LIN {X 0,Y 418.256,Z 157.888,A -85,B 0,C 180,E1 -10109.163,E2 -10109.163} C_VEL
LIN {X 0,Y 418.233,Z 157.886,A -85,B 0,C 180,E1 -10112.53,E2 -10112.53} C_VEL
LIN {X 0,Y 418.25,Z 157.887,A -85,B 0,C 180,E1 -10114.842,E2 -10114.842} C_VEL
LIN {X 0,Y 418.23,Z 157.886,A -85,B 0,C 180,E1 -10118.445,E2 -10118.445} C_VEL
LIN {X 0,Y 418.219,Z 157.887,A -85,B 0,C 180,E1 -10122.236,E2 -10122.236} C_VEL
LIN {X 0,Y 418.238,Z 157.887,A -85,B 0,C 180,E1 -10125.108,E2 -10125.108} C_VEL
LIN {X 0,Y 418.219,Z 157.886,A -85,B 0,C 180,E1 -10127.764,E2 -10127.764} C_VEL
LIN {X 0,Y 418.198,Z 157.895,A -85,B 0,C 180,E1 -10130.629,E2 -10130.629} C_VEL
LIN {X 0,Y 418.221,Z 157.886,A -85,B 0,C 180,E1 -10133.973,E2 -10133.973} C_VEL
LIN {X 0,Y 418.231,Z 157.884,A -85,B 0,C 180,E1 -10137.47,E2 -10137.47} C_VEL
LIN {X 0,Y 418.261,Z 157.886,A -85,B 0,C 180,E1 -10140.898,E2 -10140.898} C_VEL
LIN {X 0,Y 418.242,Z 157.942,A -85,B 0,C 180,E1 -10143.423,E2 -10143.423} C_VEL
LIN {X 0,Y 418.819,Z 160.686,A -85,B 0,C 180,E1 -10144.132,E2 -10144.132} C_VEL
LIN {X 0,Y 420.946,Z 171.955,A -85,B 0,C 180,E1 -10146.675,E2 -10146.675} C_VEL
LIN {X 0,Y 420.228,Z 183.952,A -85,B 0,C 180,E1 -10149.182,E2 -10149.182} C_VEL
LIN {X 0,Y 419.697,Z 193.077,A -85,B 0,C 180,E1 -10151.036,E2 -10151.036} C_VEL
LIN {X 0,Y 420.352,Z 197.644,A -85,B 0,C 180,E1 -10151.195,E2 -10151.195} C_VEL
LIN {X 0,Y 423.589,Z 218.355,A -85,B 0,C 180,E1 -10151.71,E2 -10151.71} C_VEL
LIN {X 0,Y 422.515,Z 301.675,A -85,B 0,C 180,E1 -10153.2,E2 -10153.2} C_VEL
LIN {X 0,Y 422,Z 315.355,A -85,B 0,C 180,E1 -10153.646,E2 -10153.646} C_VEL
LIN {X 0,Y 421.401,Z 328.225,A -85,B 0,C 180,E1 -10154.275,E2 -10154.275} C_VEL
LIN {X 0,Y 420.651,Z 340.778,A -85,B 0,C 180,E1 -10155.114,E2 -10155.114} C_VEL
LIN {X 0,Y 419.944,Z 352.093,A -85,B 0,C 180,E1 -10156.089,E2 -10156.089} C_VEL
LIN {X 0,Y 419.366,Z 362.073,A -85,B 0,C 180,E1 -10157.17,E2 -10157.17} C_VEL
LIN {X 0,Y 418.661,Z 371.189,A -85,B 0,C 180,E1 -10158.378,E2 -10158.378} C_VEL
LIN {X 0,Y 418.066,Z 380.082,A -85,B 0,C 180,E1 -10159.832,E2 -10159.832} C_VEL
LIN {X 0,Y 417.587,Z 387.196,A -85,B 0,C 180,E1 -10161.287,E2 -10161.287} C_VEL
LIN {X 0,Y 417.292,Z 392.868,A -85,B 0,C 180,E1 -10162.742,E2 -10162.742} C_VEL
LIN {X 0,Y 417.127,Z 397.326,A -85,B 0,C 180,E1 -10164.197,E2 -10164.197} C_VEL
LIN {X 0,Y 417.115,Z 399.677,A -85,B 0,C 180,E1 -10165.166,E2 -10165.166} C_VEL
LIN {X 0,Y 417,Z 401.592,A -85,B 0,C 180,E1 -10166.134,E2 -10166.134} C_VEL
LIN {X 0,Y 416.985,Z 403.061,A -85,B 0,C 180,E1 -10167.101,E2 -10167.101} C_VEL
LIN {X 0,Y 417.031,Z 404.093,A -85,B 0,C 180,E1 -10168.068,E2 -10168.068} C_VEL
LIN {X 0,Y 416.983,Z 404.982,A -85,B 0,C 180,E1 -10169.999,E2 -10169.999} C_VEL
LIN {X 0,Y 416.993,Z 404.811,A -85,B 0,C 180,E1 -10170.965,E2 -10170.965} C_VEL
LIN {X 0,Y 417.03,Z 404.222,A -85,B 0,C 180,E1 -10171.93,E2 -10171.93} C_VEL
LIN {X 0,Y 417,Z 401.865,A -85,B 0,C 180,E1 -10173.864,E2 -10173.864} C_VEL
LIN {X 0,Y 417.158,Z 398.955,A -85,B 0,C 180,E1 -10175.316,E2 -10175.316} C_VEL
LIN {X 0,Y 417.245,Z 395.007,A -85,B 0,C 180,E1 -10176.77,E2 -10176.77} C_VEL
LIN {X 0,Y 417.536,Z 389.923,A -85,B 0,C 180,E1 -10178.225,E2 -10178.225} C_VEL
LIN {X 0,Y 417.921,Z 383.532,A -85,B 0,C 180,E1 -10179.68,E2 -10179.68} C_VEL
LIN {X 0,Y 418.465,Z 375.535,A -85,B 0,C 180,E1 -10181.135,E2 -10181.135} C_VEL
LIN {X 0,Y 419.313,Z 365.602,A -85,B 0,C 180,E1 -10182.584,E2 -10182.584} C_VEL
LIN {X 0,Y 419.963,Z 355.585,A -85,B 0,C 180,E1 -10183.754,E2 -10183.754} C_VEL
LIN {X 0,Y 420.694,Z 344.905,A -85,B 0,C 180,E1 -10184.758,E2 -10184.758} C_VEL
LIN {X 0,Y 421.389,Z 333.667,A -85,B 0,C 180,E1 -10185.6,E2 -10185.6} C_VEL
LIN {X 0,Y 422.192,Z 321.034,A -85,B 0,C 180,E1 -10186.313,E2 -10186.313} C_VEL
LIN {X 0,Y 422.754,Z 307.58,A -85,B 0,C 180,E1 -10186.85,E2 -10186.85} C_VEL
LIN {X 0,Y 423.111,Z 294.306,A -85,B 0,C 180,E1 -10187.177,E2 -10187.177} C_VEL
LIN {X 0,Y 423.985,Z 216.483,A -85,B 0,C 180,E1 -10188.568,E2 -10188.568} C_VEL
LIN {X 0,Y 420.139,Z 194.167,A -85,B 0,C 180,E1 -10189.181,E2 -10189.181} C_VEL
LIN {X 0,Y 419.921,Z 192.559,A -85,B 0,C 180,E1 -10189.275,E2 -10189.275} C_VEL
LIN {X 0,Y 421.094,Z 174.5,A -85,B 0,C 180,E1 -10192.964,E2 -10192.964} C_VEL
LIN {X 0,Y 420.573,Z 169.022,A -85,B 0,C 180,E1 -10194.166,E2 -10194.166} C_VEL
LIN {X 0,Y 418.252,Z 157.975,A -85,B 0,C 180,E1 -10196.777,E2 -10196.777} C_VEL
LIN {X 0,Y 418.23,Z 157.89,A -85,B 0,C 180,E1 -10200.272,E2 -10200.272} C_VEL
LIN {X 0,Y 418.226,Z 157.888,A -85,B 0,C 180,E1 -10203.677,E2 -10203.677} C_VEL
LIN {X 0,Y 418.226,Z 157.891,A -85,B 0,C 180,E1 -10207.224,E2 -10207.224} C_VEL
LIN {X 0,Y 418.2,Z 157.892,A -85,B 0,C 180,E1 -10210.866,E2 -10210.866} C_VEL
LIN {X 0,Y 418.194,Z 157.892,A -85,B 0,C 180,E1 -10213.726,E2 -10213.726} C_VEL
LIN {X 0,Y 418.19,Z 157.891,A -85,B 0,C 180,E1 -10216.446,E2 -10216.446} C_VEL
LIN {X 0,Y 418.198,Z 157.892,A -85,B 0,C 180,E1 -10219.132,E2 -10219.132} C_VEL
LIN {X 0,Y 418.225,Z 157.885,A -85,B 0,C 180,E1 -10222.774,E2 -10222.774} C_VEL
LIN {X 0,Y 418.222,Z 157.884,A -85,B 0,C 180,E1 -10226.32,E2 -10226.32} C_VEL
LIN {X 0,Y 418.227,Z 157.886,A -85,B 0,C 180,E1 -10229.726,E2 -10229.726} C_VEL
LIN {X 0,Y 418.198,Z 157.889,A -85,B 0,C 180,E1 -10233.015,E2 -10233.015} C_VEL
LIN {X 0,Y 418.244,Z 157.882,A -85,B 0,C 180,E1 -10236.216,E2 -10236.216} C_VEL
LIN {X 0,Y 418.237,Z 157.885,A -85,B 0,C 180,E1 -10239.336,E2 -10239.336} C_VEL
LIN {X 0,Y 418.267,Z 157.881,A -85,B 0,C 180,E1 -10242.395,E2 -10242.395} C_VEL
LIN {X 0,Y 418.284,Z 157.878,A -85,B 0,C 180,E1 -10245.402,E2 -10245.402} C_VEL
LIN {X 0,Y 418.299,Z 157.878,A -85,B 0,C 180,E1 -10248.368,E2 -10248.368} C_VEL
LIN {X 0,Y 418.453,Z 157.86,A -85,B 0,C 180,E1 -10252.278,E2 -10252.278} C_VEL
LIN {X 0,Y 418.485,Z 157.854,A -85,B 0,C 180,E1 -10254.216,E2 -10254.216} C_VEL
LIN {X 0,Y 418.523,Z 157.85,A -85,B 0,C 180,E1 -10258.075,E2 -10258.075} C_VEL
LIN {X 0,Y 418.466,Z 157.859,A -85,B 0,C 180,E1 -10260.962,E2 -10260.962} C_VEL
LIN {X 0,Y 418.46,Z 157.856,A -85,B 0,C 180,E1 -10262.888,E2 -10262.888} C_VEL
LIN {X 0,Y 418.45,Z 157.861,A -85,B 0,C 180,E1 -10266.682,E2 -10266.682} C_VEL
LIN {X 0,Y 418.311,Z 157.875,A -85,B 0,C 180,E1 -10269.672,E2 -10269.672} C_VEL
LIN {X 0,Y 418.332,Z 157.874,A -85,B 0,C 180,E1 -10273,E2 -10273} C_VEL
LIN {X 0,Y 418.298,Z 157.881,A -85,B 0,C 180,E1 -10276.735,E2 -10276.735} C_VEL
LIN {X 0,Y 418.256,Z 157.885,A -85,B 0,C 180,E1 -10279.79,E2 -10279.79} C_VEL
LIN {X 0,Y 418.214,Z 157.891,A -85,B 0,C 180,E1 -10282.737,E2 -10282.737} C_VEL
LIN {X 0,Y 418.204,Z 157.893,A -85,B 0,C 180,E1 -10285.908,E2 -10285.908} C_VEL
LIN {X 0,Y 418.269,Z 158.07,A -85,B 0,C 180,E1 -10289.645,E2 -10289.645} C_VEL
LIN {X 0,Y 420.353,Z 168.154,A -85,B 0,C 180,E1 -10292.061,E2 -10292.061} C_VEL
LIN {X 0,Y 420.567,Z 172.653,A -85,B 0,C 180,E1 -10293.062,E2 -10293.062} C_VEL
LIN {X 0,Y 420.213,Z 181.073,A -85,B 0,C 180,E1 -10294.813,E2 -10294.813} C_VEL
LIN {X 0,Y 423.231,Z 196.278,A -85,B 0,C 180,E1 -10295.287,E2 -10295.287} C_VEL
LIN {X 0,Y 424.291,Z 202.854,A -85,B 0,C 180,E1 -10295.463,E2 -10295.463} C_VEL
LIN {X 0,Y 422.997,Z 288.987,A -85,B 0,C 180,E1 -10297.017,E2 -10297.017} C_VEL
LIN {X 0,Y 422.616,Z 302.178,A -85,B 0,C 180,E1 -10297.45,E2 -10297.45} C_VEL
LIN {X 0,Y 422.093,Z 314.233,A -85,B 0,C 180,E1 -10298.029,E2 -10298.029} C_VEL
LIN {X 0,Y 421.458,Z 325.771,A -85,B 0,C 180,E1 -10298.77,E2 -10298.77} C_VEL
LIN {X 0,Y 420.642,Z 337.831,A -85,B 0,C 180,E1 -10299.778,E2 -10299.778} C_VEL
LIN {X 0,Y 419.841,Z 348.696,A -85,B 0,C 180,E1 -10300.925,E2 -10300.925} C_VEL
LIN {X 0,Y 419.105,Z 358.292,A -85,B 0,C 180,E1 -10302.198,E2 -10302.198} C_VEL
LIN {X 0,Y 418.472,Z 366.391,A -85,B 0,C 180,E1 -10303.517,E2 -10303.517} C_VEL
LIN {X 0,Y 417.906,Z 374.069,A -85,B 0,C 180,E1 -10305.066,E2 -10305.066} C_VEL
LIN {X 0,Y 417.524,Z 380.328,A -85,B 0,C 180,E1 -10306.694,E2 -10306.694} C_VEL
LIN {X 0,Y 417.245,Z 385.249,A -85,B 0,C 180,E1 -10308.373,E2 -10308.373} C_VEL
LIN {X 0,Y 417.139,Z 387.376,A -85,B 0,C 180,E1 -10309.302,E2 -10309.302} C_VEL
LIN {X 0,Y 416.926,Z 389.978,A -85,B 0,C 180,E1 -10310.841,E2 -10310.841} C_VEL
LIN {X 0,Y 416.831,Z 391.652,A -85,B 0,C 180,E1 -10312.631,E2 -10312.631} C_VEL
LIN {X 0,Y 416.778,Z 392.031,A -85,B 0,C 180,E1 -10314.037,E2 -10314.037} C_VEL
LIN {X 0,Y 416.834,Z 391.349,A -85,B 0,C 180,E1 -10315.706,E2 -10315.706} C_VEL
LIN {X 0,Y 416.908,Z 389.362,A -85,B 0,C 180,E1 -10317.444,E2 -10317.444} C_VEL
LIN {X 0,Y 417.17,Z 385.931,A -85,B 0,C 180,E1 -10319.225,E2 -10319.225} C_VEL
LIN {X 0,Y 417.366,Z 381.677,A -85,B 0,C 180,E1 -10320.771,E2 -10320.771} C_VEL
LIN {X 0,Y 417.733,Z 375.554,A -85,B 0,C 180,E1 -10322.442,E2 -10322.442} C_VEL
LIN {X 0,Y 418.212,Z 367.784,A -85,B 0,C 180,E1 -10324.094,E2 -10324.094} C_VEL
LIN {X 0,Y 418.738,Z 359.673,A -85,B 0,C 180,E1 -10325.457,E2 -10325.457} C_VEL
LIN {X 0,Y 419.405,Z 350.387,A -85,B 0,C 180,E1 -10326.724,E2 -10326.724} C_VEL
LIN {X 0,Y 420.143,Z 339.8,A -85,B 0,C 180,E1 -10327.892,E2 -10327.892} C_VEL
LIN {X 0,Y 420.86,Z 328.814,A -85,B 0,C 180,E1 -10328.854,E2 -10328.854} C_VEL
LIN {X 0,Y 421.51,Z 316.491,A -85,B 0,C 180,E1 -10329.697,E2 -10329.697} C_VEL
LIN {X 0,Y 421.984,Z 304.982,A -85,B 0,C 180,E1 -10330.292,E2 -10330.292} C_VEL
LIN {X 0,Y 422.414,Z 292.048,A -85,B 0,C 180,E1 -10330.758,E2 -10330.758} C_VEL
LIN {X 0,Y 422.684,Z 275.71,A -85,B 0,C 180,E1 -10331.1,E2 -10331.1} C_VEL
LIN {X 0,Y 423.205,Z 232.959,A -85,B 0,C 180,E1 -10331.848,E2 -10331.848} C_VEL
LIN {X 0,Y 422.703,Z 227.158,A -85,B 0,C 180,E1 -10331.974,E2 -10331.974} C_VEL
LIN {X 0,Y 417.261,Z 206.531,A -85,B 0,C 180,E1 -10332.579,E2 -10332.579} C_VEL
LIN {X 0,Y 416.803,Z 202.658,A -85,B 0,C 180,E1 -10332.67,E2 -10332.67} C_VEL
LIN {X 0,Y 412.969,Z 181.704,A -85,B 0,C 180,E1 -10333.248,E2 -10333.248} C_VEL
LIN {X 0,Y 412.905,Z 180.585,A -85,B 0,C 180,E1 -10333.373,E2 -10333.373} C_VEL
LIN {X 0,Y 413.489,Z 170.534,A -85,B 0,C 180,E1 -10335.652,E2 -10335.652} C_VEL
LIN {X 0,Y 411.309,Z 158.9,A -85,B 0,C 180,E1 -10338.544,E2 -10338.544} C_VEL
LIN {X 0,Y 411.441,Z 158.734,A -85,B 0,C 180,E1 -10342.185,E2 -10342.185} C_VEL
LIN {X 0,Y 411.472,Z 158.731,A -85,B 0,C 180,E1 -10344.119,E2 -10344.119} C_VEL
LIN {X 0,Y 411.508,Z 158.726,A -85,B 0,C 180,E1 -10348.044,E2 -10348.044} C_VEL
LIN {X 0,Y 411.637,Z 158.71,A -85,B 0,C 180,E1 -10350.001,E2 -10350.001} C_VEL
LIN {X 0,Y 411.455,Z 158.729,A -85,B 0,C 180,E1 -10352.938,E2 -10352.938} C_VEL
LIN {X 0,Y 411.464,Z 158.731,A -85,B 0,C 180,E1 -10355.883,E2 -10355.883} C_VEL
LIN {X 0,Y 411.317,Z 158.746,A -85,B 0,C 180,E1 -10358.847,E2 -10358.847} C_VEL
LIN {X 0,Y 411.283,Z 158.753,A -85,B 0,C 180,E1 -10361.834,E2 -10361.834} C_VEL
LIN {X 0,Y 411.259,Z 158.754,A -85,B 0,C 180,E1 -10364.854,E2 -10364.854} C_VEL
LIN {X 0,Y 411.244,Z 158.756,A -85,B 0,C 180,E1 -10367.916,E2 -10367.916} C_VEL
LIN {X 0,Y 411.195,Z 158.765,A -85,B 0,C 180,E1 -10371.035,E2 -10371.035} C_VEL
LIN {X 0,Y 411.224,Z 158.757,A -85,B 0,C 180,E1 -10374.216,E2 -10374.216} C_VEL
LIN {X 0,Y 411.258,Z 158.756,A -85,B 0,C 180,E1 -10377.478,E2 -10377.478} C_VEL
LIN {X 0,Y 411.188,Z 158.766,A -85,B 0,C 180,E1 -10380.848,E2 -10380.848} C_VEL
LIN {X 0,Y 411.204,Z 158.761,A -85,B 0,C 180,E1 -10384.334,E2 -10384.334} C_VEL
LIN {X 0,Y 411.191,Z 158.761,A -85,B 0,C 180,E1 -10387.975,E2 -10387.975} C_VEL
LIN {X 0,Y 411.163,Z 158.768,A -85,B 0,C 180,E1 -10391.229,E2 -10391.229} C_VEL
LIN {X 0,Y 411.175,Z 158.767,A -85,B 0,C 180,E1 -10394.491,E2 -10394.491} C_VEL
LIN {X 0,Y 411.171,Z 158.766,A -85,B 0,C 180,E1 -10398.195,E2 -10398.195} C_VEL
LIN {X 0,Y 411.197,Z 158.766,A -85,B 0,C 180,E1 -10400.774,E2 -10400.774} C_VEL
LIN {X 0,Y 411.197,Z 158.767,A -85,B 0,C 180,E1 -10404.472,E2 -10404.472} C_VEL
LIN {X 0,Y 411.207,Z 158.762,A -85,B 0,C 180,E1 -10406.874,E2 -10406.874} C_VEL
LIN {X 0,Y 411.212,Z 158.763,A -85,B 0,C 180,E1 -10410.65,E2 -10410.65} C_VEL
LIN {X 0,Y 411.195,Z 158.761,A -85,B 0,C 180,E1 -10413.617,E2 -10413.617} C_VEL
LIN {X 0,Y 411.202,Z 158.761,A -85,B 0,C 180,E1 -10416.853,E2 -10416.853} C_VEL
LIN {X 0,Y 411.215,Z 158.763,A -85,B 0,C 180,E1 -10420.051,E2 -10420.051} C_VEL
LIN {X 0,Y 411.264,Z 158.752,A -85,B 0,C 180,E1 -10423.132,E2 -10423.132} C_VEL
LIN {X 0,Y 411.306,Z 158.747,A -85,B 0,C 180,E1 -10426.897,E2 -10426.897} C_VEL
LIN {X 0,Y 411.288,Z 158.754,A -85,B 0,C 180,E1 -10430.162,E2 -10430.162} C_VEL
LIN {X 0,Y 411.39,Z 158.737,A -85,B 0,C 180,E1 -10433.132,E2 -10433.132} C_VEL
LIN {X 0,Y 411.289,Z 158.749,A -85,B 0,C 180,E1 -10435.099,E2 -10435.099} C_VEL
LIN {X 0,Y 411.502,Z 158.727,A -85,B 0,C 180,E1 -10438.043,E2 -10438.043} C_VEL
LIN {X 0,Y 411.377,Z 158.738,A -85,B 0,C 180,E1 -10440.979,E2 -10440.979} C_VEL
LIN {X 0,Y 411.439,Z 158.731,A -85,B 0,C 180,E1 -10442.938,E2 -10442.938} C_VEL
LIN {X 0,Y 411.386,Z 158.737,A -85,B 0,C 180,E1 -10446.869,E2 -10446.869} C_VEL
LIN {X 0,Y 411.282,Z 158.754,A -85,B 0,C 180,E1 -10449.839,E2 -10449.839} C_VEL
LIN {X 0,Y 411.307,Z 158.749,A -85,B 0,C 180,E1 -10453.104,E2 -10453.104} C_VEL
LIN {X 0,Y 411.259,Z 158.754,A -85,B 0,C 180,E1 -10456.889,E2 -10456.889} C_VEL
LIN {X 0,Y 411.212,Z 158.76,A -85,B 0,C 180,E1 -10459.988,E2 -10459.988} C_VEL
LIN {X 0,Y 411.189,Z 158.767,A -85,B 0,C 180,E1 -10463.149,E2 -10463.149} C_VEL
LIN {X 0,Y 411.165,Z 158.765,A -85,B 0,C 180,E1 -10466.386,E2 -10466.386} C_VEL
LIN {X 0,Y 411.194,Z 158.762,A -85,B 0,C 180,E1 -10469.714,E2 -10469.714} C_VEL
LIN {X 0,Y 411.205,Z 158.766,A -85,B 0,C 180,E1 -10473.156,E2 -10473.156} C_VEL
LIN {X 0,Y 411.19,Z 158.764,A -85,B 0,C 180,E1 -10476.552,E2 -10476.552} C_VEL
LIN {X 0,Y 411.166,Z 158.765,A -85,B 0,C 180,E1 -10479.719,E2 -10479.719} C_VEL
LIN {X 0,Y 411.163,Z 158.768,A -85,B 0,C 180,E1 -10483.135,E2 -10483.135} C_VEL
LIN {X 0,Y 411.166,Z 158.764,A -85,B 0,C 180,E1 -10485.882,E2 -10485.882} C_VEL
LIN {X 0,Y 411.158,Z 158.766,A -85,B 0,C 180,E1 -10489.492,E2 -10489.492} C_VEL
LIN {X 0,Y 411.173,Z 158.765,A -85,B 0,C 180,E1 -10492.023,E2 -10492.023} C_VEL
LIN {X 0,Y 411.185,Z 158.764,A -85,B 0,C 180,E1 -10495.127,E2 -10495.127} C_VEL
LIN {X 0,Y 411.176,Z 158.769,A -85,B 0,C 180,E1 -10498.719,E2 -10498.719} C_VEL
LIN {X 0,Y 411.171,Z 158.769,A -85,B 0,C 180,E1 -10501.406,E2 -10501.406} C_VEL
LIN {X 0,Y 411.222,Z 158.886,A -85,B 0,C 180,E1 -10503.221,E2 -10503.221} C_VEL
LIN {X 0,Y 413.471,Z 170.32,A -85,B 0,C 180,E1 -10505.924,E2 -10505.924} C_VEL
LIN {X 0,Y 413.991,Z 173.4,A -85,B 0,C 180,E1 -10506.622,E2 -10506.622} C_VEL
LIN {X 0,Y 413.246,Z 184.945,A -85,B 0,C 180,E1 -10509.074,E2 -10509.074} C_VEL
LIN {X 0,Y 412.771,Z 193.03,A -85,B 0,C 180,E1 -10510.738,E2 -10510.738} C_VEL
LIN {X 0,Y 413.463,Z 197.805,A -85,B 0,C 180,E1 -10510.903,E2 -10510.903} C_VEL
LIN {X 0,Y 416.802,Z 218.516,A -85,B 0,C 180,E1 -10511.429,E2 -10511.429} C_VEL
LIN {X 0,Y 415.661,Z 301.815,A -85,B 0,C 180,E1 -10512.947,E2 -10512.947} C_VEL
LIN {X 0,Y 415.124,Z 315.406,A -85,B 0,C 180,E1 -10513.399,E2 -10513.399} C_VEL
LIN {X 0,Y 414.534,Z 327.718,A -85,B 0,C 180,E1 -10514.007,E2 -10514.007} C_VEL
LIN {X 0,Y 413.759,Z 340.356,A -85,B 0,C 180,E1 -10514.861,E2 -10514.861} C_VEL
LIN {X 0,Y 413.036,Z 351.734,A -85,B 0,C 180,E1 -10515.851,E2 -10515.851} C_VEL
LIN {X 0,Y 412.417,Z 361.772,A -85,B 0,C 180,E1 -10516.95,E2 -10516.95} C_VEL
LIN {X 0,Y 411.681,Z 370.921,A -85,B 0,C 180,E1 -10518.178,E2 -10518.178} C_VEL
LIN {X 0,Y 411.046,Z 379.843,A -85,B 0,C 180,E1 -10519.657,E2 -10519.657} C_VEL
LIN {X 0,Y 410.55,Z 386.991,A -85,B 0,C 180,E1 -10521.136,E2 -10521.136} C_VEL
LIN {X 0,Y 410.216,Z 392.684,A -85,B 0,C 180,E1 -10522.617,E2 -10522.617} C_VEL
LIN {X 0,Y 410.045,Z 397.16,A -85,B 0,C 180,E1 -10524.096,E2 -10524.096} C_VEL
LIN {X 0,Y 410.029,Z 399.52,A -85,B 0,C 180,E1 -10525.083,E2 -10525.083} C_VEL
LIN {X 0,Y 409.92,Z 401.444,A -85,B 0,C 180,E1 -10526.067,E2 -10526.067} C_VEL
LIN {X 0,Y 409.884,Z 402.926,A -85,B 0,C 180,E1 -10527.05,E2 -10527.05} C_VEL
LIN {X 0,Y 409.927,Z 403.966,A -85,B 0,C 180,E1 -10528.034,E2 -10528.034} C_VEL
LIN {X 0,Y 409.919,Z 404.612,A -85,B 0,C 180,E1 -10529.017,E2 -10529.017} C_VEL
LIN {X 0,Y 409.907,Z 404.868,A -85,B 0,C 180,E1 -10529.999,E2 -10529.999} C_VEL
LIN {X 0,Y 409.919,Z 404.71,A -85,B 0,C 180,E1 -10530.981,E2 -10530.981} C_VEL
LIN {X 0,Y 409.926,Z 404.126,A -85,B 0,C 180,E1 -10531.964,E2 -10531.964} C_VEL
LIN {X 0,Y 409.922,Z 401.779,A -85,B 0,C 180,E1 -10533.931,E2 -10533.931} C_VEL
LIN {X 0,Y 410.075,Z 398.879,A -85,B 0,C 180,E1 -10535.408,E2 -10535.408} C_VEL
LIN {X 0,Y 410.182,Z 394.942,A -85,B 0,C 180,E1 -10536.887,E2 -10536.887} C_VEL
LIN {X 0,Y 410.481,Z 389.869,A -85,B 0,C 180,E1 -10538.367,E2 -10538.367} C_VEL
LIN {X 0,Y 410.893,Z 383.493,A -85,B 0,C 180,E1 -10539.847,E2 -10539.847} C_VEL
LIN {X 0,Y 411.481,Z 375.511,A -85,B 0,C 180,E1 -10541.326,E2 -10541.326} C_VEL
LIN {X 0,Y 412.378,Z 365.595,A -85,B 0,C 180,E1 -10542.799,E2 -10542.799} C_VEL
LIN {X 0,Y 413.102,Z 355.019,A -85,B 0,C 180,E1 -10544.052,E2 -10544.052} C_VEL
LIN {X 0,Y 413.961,Z 343.568,A -85,B 0,C 180,E1 -10545.13,E2 -10545.13} C_VEL
LIN {X 0,Y 414.746,Z 332.01,A -85,B 0,C 180,E1 -10545.982,E2 -10545.982} C_VEL
LIN {X 0,Y 415.46,Z 320.05,A -85,B 0,C 180,E1 -10546.648,E2 -10546.648} C_VEL
LIN {X 0,Y 416.031,Z 307.184,A -85,B 0,C 180,E1 -10547.162,E2 -10547.162} C_VEL
LIN {X 0,Y 416.373,Z 293.683,A -85,B 0,C 180,E1 -10547.496,E2 -10547.496} C_VEL
LIN {X 0,Y 417.341,Z 217.423,A -85,B 0,C 180,E1 -10548.88,E2 -10548.88} C_VEL
LIN {X 0,Y 413.395,Z 194.678,A -85,B 0,C 180,E1 -10549.519,E2 -10549.519} C_VEL
LIN {X 0,Y 413.032,Z 192.431,A -85,B 0,C 180,E1 -10549.645,E2 -10549.645} C_VEL
LIN {X 0,Y 414.154,Z 176.39,A -85,B 0,C 180,E1 -10552.972,E2 -10552.972} C_VEL
LIN {X 0,Y 413.83,Z 171.504,A -85,B 0,C 180,E1 -10554.052,E2 -10554.052} C_VEL
LIN {X 0,Y 411.575,Z 160.565,A -85,B 0,C 180,E1 -10556.62,E2 -10556.62} C_VEL
LIN {X 0,Y 411.164,Z 158.798,A -85,B 0,C 180,E1 -10557.139,E2 -10557.139} C_VEL
LIN {X 0,Y 411.188,Z 158.767,A -85,B 0,C 180,E1 -10559.712,E2 -10559.712} C_VEL
LIN {X 0,Y 411.2,Z 158.762,A -85,B 0,C 180,E1 -10563.155,E2 -10563.155} C_VEL
LIN {X 0,Y 411.183,Z 158.765,A -85,B 0,C 180,E1 -10566.55,E2 -10566.55} C_VEL
LIN {X 0,Y 411.161,Z 158.769,A -85,B 0,C 180,E1 -10569.718,E2 -10569.718} C_VEL
LIN {X 0,Y 411.154,Z 158.772,A -85,B 0,C 180,E1 -10573.134,E2 -10573.134} C_VEL
LIN {X 0,Y 411.155,Z 158.769,A -85,B 0,C 180,E1 -10575.881,E2 -10575.881} C_VEL
LIN {X 0,Y 411.149,Z 158.769,A -85,B 0,C 180,E1 -10579.491,E2 -10579.491} C_VEL
LIN {X 0,Y 411.174,Z 158.762,A -85,B 0,C 180,E1 -10582.024,E2 -10582.024} C_VEL
LIN {X 0,Y 411.193,Z 158.763,A -85,B 0,C 180,E1 -10585.122,E2 -10585.122} C_VEL
LIN {X 0,Y 411.149,Z 158.767,A -85,B 0,C 180,E1 -10588.001,E2 -10588.001} C_VEL
LIN {X 0,Y 411.16,Z 158.767,A -85,B 0,C 180,E1 -10591.405,E2 -10591.405} C_VEL
LIN {X 0,Y 411.177,Z 158.77,A -85,B 0,C 180,E1 -10594.94,E2 -10594.94} C_VEL
LIN {X 0,Y 411.191,Z 158.761,A -85,B 0,C 180,E1 -10597.912,E2 -10597.912} C_VEL
LIN {X 0,Y 411.206,Z 158.759,A -85,B 0,C 180,E1 -10601.05,E2 -10601.05} C_VEL
LIN {X 0,Y 411.239,Z 158.755,A -85,B 0,C 180,E1 -10604.131,E2 -10604.131} C_VEL
LIN {X 0,Y 411.29,Z 158.752,A -85,B 0,C 180,E1 -10607.165,E2 -10607.165} C_VEL
LIN {X 0,Y 411.275,Z 158.751,A -85,B 0,C 180,E1 -10610.16,E2 -10610.16} C_VEL
LIN {X 0,Y 411.419,Z 158.734,A -85,B 0,C 180,E1 -10613.132,E2 -10613.132} C_VEL
LIN {X 0,Y 411.284,Z 158.752,A -85,B 0,C 180,E1 -10615.098,E2 -10615.098} C_VEL
LIN {X 0,Y 411.492,Z 158.725,A -85,B 0,C 180,E1 -10618.042,E2 -10618.042} C_VEL
LIN {X 0,Y 411.488,Z 158.727,A -85,B 0,C 180,E1 -10621.957,E2 -10621.957} C_VEL
LIN {X 0,Y 411.429,Z 158.734,A -85,B 0,C 180,E1 -10625.882,E2 -10625.882} C_VEL
LIN {X 0,Y 411.399,Z 158.739,A -85,B 0,C 180,E1 -10627.854,E2 -10627.854} C_VEL
LIN {X 0,Y 411.259,Z 158.755,A -85,B 0,C 180,E1 -10631.833,E2 -10631.833} C_VEL
LIN {X 0,Y 411.244,Z 158.759,A -85,B 0,C 180,E1 -10634.853,E2 -10634.853} C_VEL
LIN {X 0,Y 411.23,Z 158.761,A -85,B 0,C 180,E1 -10637.916,E2 -10637.916} C_VEL
LIN {X 0,Y 411.182,Z 158.765,A -85,B 0,C 180,E1 -10641.034,E2 -10641.034} C_VEL
LIN {X 0,Y 411.178,Z 158.769,A -85,B 0,C 180,E1 -10644.218,E2 -10644.218} C_VEL
LIN {X 0,Y 411.132,Z 158.774,A -85,B 0,C 180,E1 -10647.486,E2 -10647.486} C_VEL
LIN {X 0,Y 411.237,Z 158.997,A -85,B 0,C 180,E1 -10649.36,E2 -10649.36} C_VEL
LIN {X 0,Y 413.321,Z 169.043,A -85,B 0,C 180,E1 -10651.81,E2 -10651.81} C_VEL
LIN {X 0,Y 413.665,Z 173.968,A -85,B 0,C 180,E1 -10652.933,E2 -10652.933} C_VEL
LIN {X 0,Y 413.31,Z 181.143,A -85,B 0,C 180,E1 -10654.447,E2 -10654.447} C_VEL
LIN {X 0,Y 414.752,Z 188.124,A -85,B 0,C 180,E1 -10654.697,E2 -10654.697} C_VEL
LIN {X 0,Y 417.615,Z 203.869,A -85,B 0,C 180,E1 -10655.147,E2 -10655.147} C_VEL
LIN {X 0,Y 416.269,Z 289.366,A -85,B 0,C 180,E1 -10656.719,E2 -10656.719} C_VEL
LIN {X 0,Y 415.84,Z 302.779,A -85,B 0,C 180,E1 -10657.171,E2 -10657.171} C_VEL
LIN {X 0,Y 415.243,Z 315.436,A -85,B 0,C 180,E1 -10657.8,E2 -10657.8} C_VEL
LIN {X 0,Y 414.552,Z 327.567,A -85,B 0,C 180,E1 -10658.624,E2 -10658.624} C_VEL
LIN {X 0,Y 413.731,Z 338.588,A -85,B 0,C 180,E1 -10659.579,E2 -10659.579} C_VEL
LIN {X 0,Y 412.879,Z 349.419,A -85,B 0,C 180,E1 -10660.76,E2 -10660.76} C_VEL
LIN {X 0,Y 412.098,Z 359.283,A -85,B 0,C 180,E1 -10662.113,E2 -10662.113} C_VEL
LIN {X 0,Y 411.367,Z 367.998,A -85,B 0,C 180,E1 -10663.594,E2 -10663.594} C_VEL
LIN {X 0,Y 410.87,Z 374.556,A -85,B 0,C 180,E1 -10664.985,E2 -10664.985} C_VEL
LIN {X 0,Y 410.424,Z 381.163,A -85,B 0,C 180,E1 -10666.771,E2 -10666.771} C_VEL
LIN {X 0,Y 410.149,Z 386.065,A -85,B 0,C 180,E1 -10668.544,E2 -10668.544} C_VEL
LIN {X 0,Y 410.034,Z 387.794,A -85,B 0,C 180,E1 -10669.361,E2 -10669.361} C_VEL
LIN {X 0,Y 409.848,Z 389.877,A -85,B 0,C 180,E1 -10670.621,E2 -10670.621} C_VEL
LIN {X 0,Y 409.744,Z 391.438,A -85,B 0,C 180,E1 -10672.091,E2 -10672.091} C_VEL
LIN {X 0,Y 409.681,Z 392.125,A -85,B 0,C 180,E1 -10673.733,E2 -10673.733} C_VEL
LIN {X 0,Y 409.724,Z 391.611,A -85,B 0,C 180,E1 -10675.527,E2 -10675.527} C_VEL
LIN {X 0,Y 409.78,Z 389.922,A -85,B 0,C 180,E1 -10677.18,E2 -10677.18} C_VEL
LIN {X 0,Y 410.061,Z 386.548,A -85,B 0,C 180,E1 -10679.06,E2 -10679.06} C_VEL
LIN {X 0,Y 410.292,Z 381.746,A -85,B 0,C 180,E1 -10680.878,E2 -10680.878} C_VEL
LIN {X 0,Y 410.655,Z 376.011,A -85,B 0,C 180,E1 -10682.48,E2 -10682.48} C_VEL
LIN {X 0,Y 411.166,Z 368.308,A -85,B 0,C 180,E1 -10684.161,E2 -10684.161} C_VEL
LIN {X 0,Y 411.717,Z 360.317,A -85,B 0,C 180,E1 -10685.549,E2 -10685.549} C_VEL
LIN {X 0,Y 412.467,Z 350.309,A -85,B 0,C 180,E1 -10686.94,E2 -10686.94} C_VEL
LIN {X 0,Y 413.147,Z 340.685,A -85,B 0,C 180,E1 -10688.024,E2 -10688.024} C_VEL
LIN {X 0,Y 413.934,Z 329.496,A -85,B 0,C 180,E1 -10689.037,E2 -10689.037} C_VEL
LIN {X 0,Y 414.532,Z 317.928,A -85,B 0,C 180,E1 -10689.857,E2 -10689.857} C_VEL
LIN {X 0,Y 415.113,Z 305.328,A -85,B 0,C 180,E1 -10690.532,E2 -10690.532} C_VEL
LIN {X 0,Y 415.567,Z 292.382,A -85,B 0,C 180,E1 -10691.011,E2 -10691.011} C_VEL
LIN {X 0,Y 415.879,Z 277.35,A -85,B 0,C 180,E1 -10691.335,E2 -10691.335} C_VEL
LIN {X 0,Y 416.803,Z 202.658,A -85,B 0,C 180,E1 -10692.67,E2 -10692.67} C_VEL
LIN {X 0,Y 415.772,Z 198.953,A -85,B 0,C 180,E1 -10692.784,E2 -10692.784} C_VEL
LIN {X 0,Y 412.048,Z 193.684,A -85,B 0,C 180,E1 -10693.047,E2 -10693.047} C_VEL
LIN {X 0,Y 408.051,Z 188.481,A -85,B 0,C 180,E1 -10693.326,E2 -10693.326} C_VEL
LIN {X 0,Y 406.621,Z 184.833,A -85,B 0,C 180,E1 -10693.461,E2 -10693.461} C_VEL
LIN {X 0,Y 405.979,Z 181.253,A -85,B 0,C 180,E1 -10693.598,E2 -10693.598} C_VEL
LIN {X 0,Y 406.494,Z 172.767,A -85,B 0,C 180,E1 -10695.51,E2 -10695.51} C_VEL
LIN {X 0,Y 405.255,Z 164.782,A -85,B 0,C 180,E1 -10697.481,E2 -10697.481} C_VEL
LIN {X 0,Y 404.243,Z 159.662,A -85,B 0,C 180,E1 -10698.849,E2 -10698.849} C_VEL
LIN {X 0,Y 404.403,Z 159.611,A -85,B 0,C 180,E1 -10702.128,E2 -10702.128} C_VEL
LIN {X 0,Y 404.42,Z 159.61,A -85,B 0,C 180,E1 -10704.016,E2 -10704.016} C_VEL
LIN {X 0,Y 404.477,Z 159.602,A -85,B 0,C 180,E1 -10708.01,E2 -10708.01} C_VEL
LIN {X 0,Y 404.607,Z 159.586,A -85,B 0,C 180,E1 -10710.001,E2 -10710.001} C_VEL
LIN {X 0,Y 404.414,Z 159.606,A -85,B 0,C 180,E1 -10712.989,E2 -10712.989} C_VEL
LIN {X 0,Y 404.411,Z 159.609,A -85,B 0,C 180,E1 -10715.986,E2 -10715.986} C_VEL
LIN {X 0,Y 404.264,Z 159.626,A -85,B 0,C 180,E1 -10719.003,E2 -10719.003} C_VEL
LIN {X 0,Y 404.255,Z 159.627,A -85,B 0,C 180,E1 -10722.042,E2 -10722.042} C_VEL
LIN {X 0,Y 404.205,Z 159.635,A -85,B 0,C 180,E1 -10725.119,E2 -10725.119} C_VEL
LIN {X 0,Y 404.203,Z 159.632,A -85,B 0,C 180,E1 -10728.239,E2 -10728.239} C_VEL
LIN {X 0,Y 404.138,Z 159.645,A -85,B 0,C 180,E1 -10731.42,E2 -10731.42} C_VEL
LIN {X 0,Y 404.175,Z 159.637,A -85,B 0,C 180,E1 -10734.666,E2 -10734.666} C_VEL
LIN {X 0,Y 404.194,Z 159.633,A -85,B 0,C 180,E1 -10738,E2 -10738} C_VEL
LIN {X 0,Y 404.138,Z 159.642,A -85,B 0,C 180,E1 -10741.559,E2 -10741.559} C_VEL
LIN {X 0,Y 404.183,Z 159.641,A -85,B 0,C 180,E1 -10745.017,E2 -10745.017} C_VEL
LIN {X 0,Y 404.15,Z 159.644,A -85,B 0,C 180,E1 -10748.758,E2 -10748.758} C_VEL
LIN {X 0,Y 404.122,Z 159.642,A -85,B 0,C 180,E1 -10751.6,E2 -10751.6} C_VEL
LIN {X 0,Y 404.145,Z 159.643,A -85,B 0,C 180,E1 -10754.523,E2 -10754.523} C_VEL
LIN {X 0,Y 404.132,Z 159.642,A -85,B 0,C 180,E1 -10757.296,E2 -10757.296} C_VEL
LIN {X 0,Y 404.132,Z 159.641,A -85,B 0,C 180,E1 -10759.952,E2 -10759.952} C_VEL
LIN {X 0,Y 404.134,Z 159.642,A -85,B 0,C 180,E1 -10763.126,E2 -10763.126} C_VEL
LIN {X 0,Y 404.145,Z 159.642,A -85,B 0,C 180,E1 -10766.188,E2 -10766.188} C_VEL
LIN {X 0,Y 404.144,Z 159.64,A -85,B 0,C 180,E1 -10769.715,E2 -10769.715} C_VEL
LIN {X 0,Y 404.134,Z 159.641,A -85,B 0,C 180,E1 -10773.119,E2 -10773.119} C_VEL
LIN {X 0,Y 404.165,Z 159.642,A -85,B 0,C 180,E1 -10776.426,E2 -10776.426} C_VEL
LIN {X 0,Y 404.192,Z 159.636,A -85,B 0,C 180,E1 -10779.875,E2 -10779.875} C_VEL
LIN {X 0,Y 404.217,Z 159.63,A -85,B 0,C 180,E1 -10782.994,E2 -10782.994} C_VEL
LIN {X 0,Y 404.284,Z 159.622,A -85,B 0,C 180,E1 -10786.939,E2 -10786.939} C_VEL
LIN {X 0,Y 404.254,Z 159.633,A -85,B 0,C 180,E1 -10789.989,E2 -10789.989} C_VEL
LIN {X 0,Y 404.341,Z 159.615,A -85,B 0,C 180,E1 -10793.012,E2 -10793.012} C_VEL
LIN {X 0,Y 404.261,Z 159.625,A -85,B 0,C 180,E1 -10795.014,E2 -10795.014} C_VEL
LIN {X 0,Y 404.471,Z 159.603,A -85,B 0,C 180,E1 -10798.009,E2 -10798.009} C_VEL
LIN {X 0,Y 404.348,Z 159.614,A -85,B 0,C 180,E1 -10800.996,E2 -10800.996} C_VEL
LIN {X 0,Y 404.398,Z 159.608,A -85,B 0,C 180,E1 -10802.989,E2 -10802.989} C_VEL
LIN {X 0,Y 404.337,Z 159.616,A -85,B 0,C 180,E1 -10806.989,E2 -10806.989} C_VEL
LIN {X 0,Y 404.249,Z 159.628,A -85,B 0,C 180,E1 -10810.012,E2 -10810.012} C_VEL
LIN {X 0,Y 404.269,Z 159.627,A -85,B 0,C 180,E1 -10813.212,E2 -10813.212} C_VEL
LIN {X 0,Y 404.218,Z 159.632,A -85,B 0,C 180,E1 -10817.007,E2 -10817.007} C_VEL
LIN {X 0,Y 404.157,Z 159.637,A -85,B 0,C 180,E1 -10820.352,E2 -10820.352} C_VEL
LIN {X 0,Y 404.15,Z 159.642,A -85,B 0,C 180,E1 -10823.576,E2 -10823.576} C_VEL
LIN {X 0,Y 404.098,Z 159.648,A -85,B 0,C 180,E1 -10826.885,E2 -10826.885} C_VEL
LIN {X 0,Y 404.141,Z 159.64,A -85,B 0,C 180,E1 -10830.286,E2 -10830.286} C_VEL
LIN {X 0,Y 404.138,Z 159.64,A -85,B 0,C 180,E1 -10833.813,E2 -10833.813} C_VEL
LIN {X 0,Y 404.133,Z 159.646,A -85,B 0,C 180,E1 -10836.874,E2 -10836.874} C_VEL
LIN {X 0,Y 404.12,Z 159.642,A -85,B 0,C 180,E1 -10840.075,E2 -10840.075} C_VEL
LIN {X 0,Y 404.143,Z 159.644,A -85,B 0,C 180,E1 -10843.082,E2 -10843.082} C_VEL
LIN {X 0,Y 404.122,Z 159.642,A -85,B 0,C 180,E1 -10845.922,E2 -10845.922} C_VEL
LIN {X 0,Y 404.103,Z 159.65,A -85,B 0,C 180,E1 -10848.632,E2 -10848.632} C_VEL
LIN {X 0,Y 404.131,Z 159.641,A -85,B 0,C 180,E1 -10851.497,E2 -10851.497} C_VEL
LIN {X 0,Y 404.157,Z 159.64,A -85,B 0,C 180,E1 -10854.98,E2 -10854.98} C_VEL
LIN {X 0,Y 404.135,Z 159.647,A -85,B 0,C 180,E1 -10858.552,E2 -10858.552} C_VEL
LIN {X 0,Y 404.15,Z 159.645,A -85,B 0,C 180,E1 -10860.862,E2 -10860.862} C_VEL
LIN {X 0,Y 404.177,Z 159.871,A -85,B 0,C 180,E1 -10863.021,E2 -10863.021} C_VEL
LIN {X 0,Y 406.402,Z 171.106,A -85,B 0,C 180,E1 -10865.704,E2 -10865.704} C_VEL
LIN {X 0,Y 407.028,Z 174.995,A -85,B 0,C 180,E1 -10866.6,E2 -10866.6} C_VEL
LIN {X 0,Y 406.206,Z 186.629,A -85,B 0,C 180,E1 -10869.114,E2 -10869.114} C_VEL
LIN {X 0,Y 405.85,Z 192.987,A -85,B 0,C 180,E1 -10870.428,E2 -10870.428} C_VEL
LIN {X 0,Y 406.676,Z 198.432,A -85,B 0,C 180,E1 -10870.613,E2 -10870.613} C_VEL
LIN {X 0,Y 409.993,Z 219.604,A -85,B 0,C 180,E1 -10871.159,E2 -10871.159} C_VEL
LIN {X 0,Y 408.842,Z 300.827,A -85,B 0,C 180,E1 -10872.653,E2 -10872.653} C_VEL
LIN {X 0,Y 408.305,Z 314.701,A -85,B 0,C 180,E1 -10873.114,E2 -10873.114} C_VEL
LIN {X 0,Y 407.679,Z 327.191,A -85,B 0,C 180,E1 -10873.731,E2 -10873.731} C_VEL
LIN {X 0,Y 406.986,Z 338.346,A -85,B 0,C 180,E1 -10874.474,E2 -10874.474} C_VEL
LIN {X 0,Y 406.208,Z 349.968,A -85,B 0,C 180,E1 -10875.471,E2 -10875.471} C_VEL
LIN {X 0,Y 405.457,Z 360.428,A -85,B 0,C 180,E1 -10876.594,E2 -10876.594} C_VEL
LIN {X 0,Y 404.843,Z 368.982,A -85,B 0,C 180,E1 -10877.721,E2 -10877.721} C_VEL
LIN {X 0,Y 404.067,Z 378.235,A -85,B 0,C 180,E1 -10879.223,E2 -10879.223} C_VEL
LIN {X 0,Y 403.564,Z 385.673,A -85,B 0,C 180,E1 -10880.729,E2 -10880.729} C_VEL
LIN {X 0,Y 403.163,Z 392.5,A -85,B 0,C 180,E1 -10882.487,E2 -10882.487} C_VEL
LIN {X 0,Y 402.947,Z 396.994,A -85,B 0,C 180,E1 -10883.992,E2 -10883.992} C_VEL
LIN {X 0,Y 402.942,Z 399.363,A -85,B 0,C 180,E1 -10884.996,E2 -10884.996} C_VEL
LIN {X 0,Y 402.842,Z 401.295,A -85,B 0,C 180,E1 -10885.997,E2 -10885.997} C_VEL
LIN {X 0,Y 402.786,Z 402.792,A -85,B 0,C 180,E1 -10886.998,E2 -10886.998} C_VEL
LIN {X 0,Y 402.824,Z 403.839,A -85,B 0,C 180,E1 -10887.999,E2 -10887.999} C_VEL
LIN {X 0,Y 402.846,Z 404.492,A -85,B 0,C 180,E1 -10888.999,E2 -10888.999} C_VEL
LIN {X 0,Y 402.833,Z 404.754,A -85,B 0,C 180,E1 -10889.999,E2 -10889.999} C_VEL
LIN {X 0,Y 402.846,Z 404.608,A -85,B 0,C 180,E1 -10890.999,E2 -10890.999} C_VEL
LIN {X 0,Y 402.823,Z 404.03,A -85,B 0,C 180,E1 -10891.999,E2 -10891.999} C_VEL
LIN {X 0,Y 402.845,Z 401.693,A -85,B 0,C 180,E1 -10894,E2 -10894} C_VEL
LIN {X 0,Y 402.972,Z 398.804,A -85,B 0,C 180,E1 -10895.503,E2 -10895.503} C_VEL
LIN {X 0,Y 403.106,Z 394.877,A -85,B 0,C 180,E1 -10897.009,E2 -10897.009} C_VEL
LIN {X 0,Y 403.441,Z 389.819,A -85,B 0,C 180,E1 -10898.514,E2 -10898.514} C_VEL
LIN {X 0,Y 403.875,Z 383.468,A -85,B 0,C 180,E1 -10900.02,E2 -10900.02} C_VEL
LIN {X 0,Y 404.507,Z 375.518,A -85,B 0,C 180,E1 -10901.524,E2 -10901.524} C_VEL
LIN {X 0,Y 405.268,Z 367.426,A -85,B 0,C 180,E1 -10902.773,E2 -10902.773} C_VEL
LIN {X 0,Y 406.017,Z 357.566,A -85,B 0,C 180,E1 -10904.023,E2 -10904.023} C_VEL
LIN {X 0,Y 406.862,Z 346.547,A -85,B 0,C 180,E1 -10905.144,E2 -10905.144} C_VEL
LIN {X 0,Y 407.764,Z 334.006,A -85,B 0,C 180,E1 -10906.135,E2 -10906.135} C_VEL
LIN {X 0,Y 408.622,Z 321.656,A -85,B 0,C 180,E1 -10906.871,E2 -10906.871} C_VEL
LIN {X 0,Y 409.243,Z 308.588,A -85,B 0,C 180,E1 -10907.424,E2 -10907.424} C_VEL
LIN {X 0,Y 409.666,Z 294.74,A -85,B 0,C 180,E1 -10907.792,E2 -10907.792} C_VEL
LIN {X 0,Y 410.666,Z 218.209,A -85,B 0,C 180,E1 -10909.208,E2 -10909.208} C_VEL
LIN {X 0,Y 406.89,Z 196.381,A -85,B 0,C 180,E1 -10909.842,E2 -10909.842} C_VEL
LIN {X 0,Y 406.179,Z 192.431,A -85,B 0,C 180,E1 -10910.009,E2 -10910.009} C_VEL
LIN {X 0,Y 407.299,Z 176.435,A -85,B 0,C 180,E1 -10913.381,E2 -10913.381} C_VEL
LIN {X 0,Y 406.195,Z 169.112,A -85,B 0,C 180,E1 -10915.079,E2 -10915.079} C_VEL
LIN {X 0,Y 404.117,Z 159.759,A -85,B 0,C 180,E1 -10917.404,E2 -10917.404} C_VEL
LIN {X 0,Y 404.136,Z 159.646,A -85,B 0,C 180,E1 -10920.284,E2 -10920.284} C_VEL
LIN {X 0,Y 404.133,Z 159.644,A -85,B 0,C 180,E1 -10923.812,E2 -10923.812} C_VEL
LIN {X 0,Y 404.125,Z 159.645,A -85,B 0,C 180,E1 -10926.872,E2 -10926.872} C_VEL
LIN {X 0,Y 404.111,Z 159.646,A -85,B 0,C 180,E1 -10930.073,E2 -10930.073} C_VEL
LIN {X 0,Y 404.134,Z 159.646,A -85,B 0,C 180,E1 -10933.08,E2 -10933.08} C_VEL
LIN {X 0,Y 404.112,Z 159.646,A -85,B 0,C 180,E1 -10935.92,E2 -10935.92} C_VEL
LIN {X 0,Y 404.093,Z 159.649,A -85,B 0,C 180,E1 -10938.631,E2 -10938.631} C_VEL
LIN {X 0,Y 404.129,Z 159.643,A -85,B 0,C 180,E1 -10941.494,E2 -10941.494} C_VEL
LIN {X 0,Y 404.164,Z 159.64,A -85,B 0,C 180,E1 -10944.981,E2 -10944.981} C_VEL
LIN {X 0,Y 404.124,Z 159.643,A -85,B 0,C 180,E1 -10948.442,E2 -10948.442} C_VEL
LIN {X 0,Y 404.138,Z 159.645,A -85,B 0,C 180,E1 -10950.861,E2 -10950.861} C_VEL
LIN {X 0,Y 404.141,Z 159.644,A -85,B 0,C 180,E1 -10954.722,E2 -10954.722} C_VEL
LIN {X 0,Y 404.154,Z 159.639,A -85,B 0,C 180,E1 -10957.507,E2 -10957.507} C_VEL
LIN {X 0,Y 404.15,Z 159.637,A -85,B 0,C 180,E1 -10960.706,E2 -10960.706} C_VEL
LIN {X 0,Y 404.207,Z 159.63,A -85,B 0,C 180,E1 -10963.847,E2 -10963.847} C_VEL
LIN {X 0,Y 404.271,Z 159.628,A -85,B 0,C 180,E1 -10966.938,E2 -10966.938} C_VEL
LIN {X 0,Y 404.241,Z 159.627,A -85,B 0,C 180,E1 -10969.987,E2 -10969.987} C_VEL
LIN {X 0,Y 404.369,Z 159.611,A -85,B 0,C 180,E1 -10973.012,E2 -10973.012} C_VEL
LIN {X 0,Y 404.256,Z 159.628,A -85,B 0,C 180,E1 -10975.013,E2 -10975.013} C_VEL
LIN {X 0,Y 404.461,Z 159.601,A -85,B 0,C 180,E1 -10978.008,E2 -10978.008} C_VEL
LIN {X 0,Y 404.457,Z 159.603,A -85,B 0,C 180,E1 -10981.991,E2 -10981.991} C_VEL
LIN {X 0,Y 404.358,Z 159.614,A -85,B 0,C 180,E1 -10986.687,E2 -10986.687} C_VEL
LIN {X 0,Y 404.231,Z 159.631,A -85,B 0,C 180,E1 -10990.012,E2 -10990.012} C_VEL
LIN {X 0,Y 404.253,Z 159.628,A -85,B 0,C 180,E1 -10993.211,E2 -10993.211} C_VEL
LIN {X 0,Y 404.203,Z 159.635,A -85,B 0,C 180,E1 -10997.007,E2 -10997.007} C_VEL
LIN {X 0,Y 404.15,Z 159.645,A -85,B 0,C 180,E1 -11000.352,E2 -11000.352} C_VEL
LIN {X 0,Y 404.136,Z 159.645,A -85,B 0,C 180,E1 -11003.576,E2 -11003.576} C_VEL
LIN {X 0,Y 404.089,Z 159.649,A -85,B 0,C 180,E1 -11006.884,E2 -11006.884} C_VEL
LIN {X 0,Y 404.189,Z 159.762,A -85,B 0,C 180,E1 -11008.991,E2 -11008.991} C_VEL
LIN {X 0,Y 406.071,Z 168.832,A -85,B 0,C 180,E1 -11011.279,E2 -11011.279} C_VEL
LIN {X 0,Y 406.809,Z 173.442,A -85,B 0,C 180,E1 -11012.381,E2 -11012.381} C_VEL
LIN {X 0,Y 406.45,Z 181.311,A -85,B 0,C 180,E1 -11014.079,E2 -11014.079} C_VEL
LIN {X 0,Y 410.479,Z 201.323,A -85,B 0,C 180,E1 -11014.726,E2 -11014.726} C_VEL
LIN {X 0,Y 410.94,Z 205.863,A -85,B 0,C 180,E1 -11014.838,E2 -11014.838} C_VEL
LIN {X 0,Y 409.564,Z 289.215,A -85,B 0,C 180,E1 -11016.396,E2 -11016.396} C_VEL
LIN {X 0,Y 409.128,Z 302.819,A -85,B 0,C 180,E1 -11016.86,E2 -11016.86} C_VEL
LIN {X 0,Y 408.461,Z 315.697,A -85,B 0,C 180,E1 -11017.51,E2 -11017.51} C_VEL
LIN {X 0,Y 407.744,Z 327.854,A -85,B 0,C 180,E1 -11018.353,E2 -11018.353} C_VEL
LIN {X 0,Y 406.858,Z 339.044,A -85,B 0,C 180,E1 -11019.341,E2 -11019.341} C_VEL
LIN {X 0,Y 406.039,Z 348.666,A -85,B 0,C 180,E1 -11020.399,E2 -11020.399} C_VEL
LIN {X 0,Y 405.201,Z 358.692,A -85,B 0,C 180,E1 -11021.774,E2 -11021.774} C_VEL
LIN {X 0,Y 404.521,Z 366.778,A -85,B 0,C 180,E1 -11023.142,E2 -11023.142} C_VEL
LIN {X 0,Y 403.83,Z 374.554,A -85,B 0,C 180,E1 -11024.777,E2 -11024.777} C_VEL
LIN {X 0,Y 403.391,Z 380.831,A -85,B 0,C 180,E1 -11026.486,E2 -11026.486} C_VEL
LIN {X 0,Y 403.16,Z 384.753,A -85,B 0,C 180,E1 -11027.847,E2 -11027.847} C_VEL
LIN {X 0,Y 402.855,Z 388.87,A -85,B 0,C 180,E1 -11029.8,E2 -11029.8} C_VEL
LIN {X 0,Y 402.684,Z 391.324,A -85,B 0,C 180,E1 -11031.755,E2 -11031.755} C_VEL
LIN {X 0,Y 402.581,Z 392.218,A -85,B 0,C 180,E1 -11033.593,E2 -11033.593} C_VEL
LIN {X 0,Y 402.605,Z 391.929,A -85,B 0,C 180,E1 -11035.129,E2 -11035.129} C_VEL
LIN {X 0,Y 402.683,Z 390.422,A -85,B 0,C 180,E1 -11036.901,E2 -11036.901} C_VEL
LIN {X 0,Y 402.925,Z 387.52,A -85,B 0,C 180,E1 -11038.723,E2 -11038.723} C_VEL
LIN {X 0,Y 403.111,Z 384.144,A -85,B 0,C 180,E1 -11040.176,E2 -11040.176} C_VEL
LIN {X 0,Y 403.419,Z 378.615,A -85,B 0,C 180,E1 -11041.943,E2 -11041.943} C_VEL
LIN {X 0,Y 403.892,Z 371.603,A -85,B 0,C 180,E1 -11043.66,E2 -11043.66} C_VEL
LIN {X 0,Y 404.414,Z 364.616,A -85,B 0,C 180,E1 -11045.024,E2 -11045.024} C_VEL
LIN {X 0,Y 405.095,Z 355.334,A -85,B 0,C 180,E1 -11046.484,E2 -11046.484} C_VEL
LIN {X 0,Y 405.905,Z 345.376,A -85,B 0,C 180,E1 -11047.745,E2 -11047.745} C_VEL
LIN {X 0,Y 406.716,Z 334.344,A -85,B 0,C 180,E1 -11048.865,E2 -11048.865} C_VEL
LIN {X 0,Y 407.441,Z 322.318,A -85,B 0,C 180,E1 -11049.821,E2 -11049.821} C_VEL
LIN {X 0,Y 408.083,Z 309.907,A -85,B 0,C 180,E1 -11050.575,E2 -11050.575} C_VEL
LIN {X 0,Y 408.625,Z 297.099,A -85,B 0,C 180,E1 -11051.125,E2 -11051.125} C_VEL
LIN {X 0,Y 409,Z 283.69,A -85,B 0,C 180,E1 -11051.491,E2 -11051.491} C_VEL
LIN {X 0,Y 410.007,Z 203.006,A -85,B 0,C 180,E1 -11052.963,E2 -11052.963} C_VEL
LIN {X 0,Y 406.621,Z 184.833,A -85,B 0,C 180,E1 -11053.461,E2 -11053.461} C_VEL
LIN {X 0,Y 405.854,Z 182.194,A -85,B 0,C 180,E1 -11053.629,E2 -11053.629} C_VEL
LIN {X 0,Y 404.399,Z 179.403,A -85,B 0,C 180,E1 -11054.057,E2 -11054.057} C_VEL
LIN {X 0,Y 400.936,Z 174.461,A -85,B 0,C 180,E1 -11055.447,E2 -11055.447} C_VEL
LIN {X 0,Y 399.137,Z 170.177,A -85,B 0,C 180,E1 -11056.552,E2 -11056.552} C_VEL
LIN {X 0,Y 398.623,Z 167.948,A -85,B 0,C 180,E1 -11057.11,E2 -11057.11} C_VEL
LIN {X 0,Y 397.226,Z 160.56,A -85,B 0,C 180,E1 -11059.069,E2 -11059.069} C_VEL
LIN {X 0,Y 397.351,Z 160.485,A -85,B 0,C 180,E1 -11062.889,E2 -11062.889} C_VEL
LIN {X 0,Y 397.251,Z 160.498,A -85,B 0,C 180,E1 -11064.926,E2 -11064.926} C_VEL
LIN {X 0,Y 397.446,Z 160.478,A -85,B 0,C 180,E1 -11067.974,E2 -11067.974} C_VEL
LIN {X 0,Y 397.576,Z 160.461,A -85,B 0,C 180,E1 -11070.001,E2 -11070.001} C_VEL
LIN {X 0,Y 397.373,Z 160.484,A -85,B 0,C 180,E1 -11073.042,E2 -11073.042} C_VEL
LIN {X 0,Y 397.362,Z 160.486,A -85,B 0,C 180,E1 -11076.093,E2 -11076.093} C_VEL
LIN {X 0,Y 397.234,Z 160.503,A -85,B 0,C 180,E1 -11079.163,E2 -11079.163} C_VEL
LIN {X 0,Y 397.218,Z 160.502,A -85,B 0,C 180,E1 -11082.259,E2 -11082.259} C_VEL
LIN {X 0,Y 397.178,Z 160.514,A -85,B 0,C 180,E1 -11085.393,E2 -11085.393} C_VEL
LIN {X 0,Y 397.157,Z 160.51,A -85,B 0,C 180,E1 -11088.575,E2 -11088.575} C_VEL
LIN {X 0,Y 397.096,Z 160.519,A -85,B 0,C 180,E1 -11091.819,E2 -11091.819} C_VEL
LIN {X 0,Y 397.155,Z 160.516,A -85,B 0,C 180,E1 -11095.132,E2 -11095.132} C_VEL
LIN {X 0,Y 397.161,Z 160.51,A -85,B 0,C 180,E1 -11097.777,E2 -11097.777} C_VEL
LIN {X 0,Y 397.078,Z 160.524,A -85,B 0,C 180,E1 -11100.883,E2 -11100.883} C_VEL
LIN {X 0,Y 397.124,Z 160.515,A -85,B 0,C 180,E1 -11104.494,E2 -11104.494} C_VEL
LIN {X 0,Y 397.099,Z 160.518,A -85,B 0,C 180,E1 -11108.276,E2 -11108.276} C_VEL
LIN {X 0,Y 397.088,Z 160.525,A -85,B 0,C 180,E1 -11110.909,E2 -11110.909} C_VEL
LIN {X 0,Y 397.1,Z 160.517,A -85,B 0,C 180,E1 -11113.649,E2 -11113.649} C_VEL
LIN {X 0,Y 397.1,Z 160.521,A -85,B 0,C 180,E1 -11116.522,E2 -11116.522} C_VEL
LIN {X 0,Y 397.088,Z 160.522,A -85,B 0,C 180,E1 -11120.42,E2 -11120.42} C_VEL
LIN {X 0,Y 397.096,Z 160.52,A -85,B 0,C 180,E1 -11123.005,E2 -11123.005} C_VEL
LIN {X 0,Y 397.118,Z 160.519,A -85,B 0,C 180,E1 -11126.283,E2 -11126.283} C_VEL
LIN {X 0,Y 397.1,Z 160.52,A -85,B 0,C 180,E1 -11130.137,E2 -11130.137} C_VEL
LIN {X 0,Y 397.095,Z 160.518,A -85,B 0,C 180,E1 -11133.739,E2 -11133.739} C_VEL
LIN {X 0,Y 397.108,Z 160.516,A -85,B 0,C 180,E1 -11137.086,E2 -11137.086} C_VEL
LIN {X 0,Y 397.148,Z 160.516,A -85,B 0,C 180,E1 -11140.353,E2 -11140.353} C_VEL
LIN {X 0,Y 397.166,Z 160.51,A -85,B 0,C 180,E1 -11143.554,E2 -11143.554} C_VEL
LIN {X 0,Y 397.23,Z 160.501,A -85,B 0,C 180,E1 -11146.703,E2 -11146.703} C_VEL
LIN {X 0,Y 397.215,Z 160.507,A -85,B 0,C 180,E1 -11149.809,E2 -11149.809} C_VEL
LIN {X 0,Y 397.293,Z 160.493,A -85,B 0,C 180,E1 -11152.887,E2 -11152.887} C_VEL
LIN {X 0,Y 397.232,Z 160.5,A -85,B 0,C 180,E1 -11154.925,E2 -11154.925} C_VEL
LIN {X 0,Y 397.44,Z 160.48,A -85,B 0,C 180,E1 -11157.974,E2 -11157.974} C_VEL
LIN {X 0,Y 397.444,Z 160.477,A -85,B 0,C 180,E1 -11162.027,E2 -11162.027} C_VEL
LIN {X 0,Y 397.317,Z 160.492,A -85,B 0,C 180,E1 -11166.093,E2 -11166.093} C_VEL
LIN {X 0,Y 397.23,Z 160.503,A -85,B 0,C 180,E1 -11169.163,E2 -11169.163} C_VEL
LIN {X 0,Y 397.219,Z 160.502,A -85,B 0,C 180,E1 -11172.259,E2 -11172.259} C_VEL
LIN {X 0,Y 397.176,Z 160.514,A -85,B 0,C 180,E1 -11175.393,E2 -11175.393} C_VEL
LIN {X 0,Y 397.157,Z 160.51,A -85,B 0,C 180,E1 -11178.574,E2 -11178.574} C_VEL
LIN {X 0,Y 397.096,Z 160.519,A -85,B 0,C 180,E1 -11181.819,E2 -11181.819} C_VEL
LIN {X 0,Y 397.103,Z 160.522,A -85,B 0,C 180,E1 -11185.136,E2 -11185.136} C_VEL
LIN {X 0,Y 397.062,Z 160.522,A -85,B 0,C 180,E1 -11188.549,E2 -11188.549} C_VEL
LIN {X 0,Y 397.076,Z 160.52,A -85,B 0,C 180,E1 -11191.835,E2 -11191.835} C_VEL
LIN {X 0,Y 397.117,Z 160.516,A -85,B 0,C 180,E1 -11194.495,E2 -11194.495} C_VEL
LIN {X 0,Y 397.089,Z 160.519,A -85,B 0,C 180,E1 -11198.277,E2 -11198.277} C_VEL
LIN {X 0,Y 397.048,Z 160.53,A -85,B 0,C 180,E1 -11200.914,E2 -11200.914} C_VEL
LIN {X 0,Y 397.089,Z 160.518,A -85,B 0,C 180,E1 -11203.651,E2 -11203.651} C_VEL
LIN {X 0,Y 397.093,Z 160.522,A -85,B 0,C 180,E1 -11206.523,E2 -11206.523} C_VEL
LIN {X 0,Y 397.086,Z 160.522,A -85,B 0,C 180,E1 -11210.419,E2 -11210.419} C_VEL
LIN {X 0,Y 397.088,Z 160.521,A -85,B 0,C 180,E1 -11213.003,E2 -11213.003} C_VEL
LIN {X 0,Y 397.09,Z 160.522,A -85,B 0,C 180,E1 -11216.289,E2 -11216.289} C_VEL
LIN {X 0,Y 397.073,Z 160.525,A -85,B 0,C 180,E1 -11219.116,E2 -11219.116} C_VEL
LIN {X 0,Y 397.061,Z 160.527,A -85,B 0,C 180,E1 -11222.253,E2 -11222.253} C_VEL
LIN {X 0,Y 397.101,Z 160.692,A -85,B 0,C 180,E1 -11222.745,E2 -11222.745} C_VEL
LIN {X 0,Y 399.441,Z 172.299,A -85,B 0,C 180,E1 -11225.577,E2 -11225.577} C_VEL
LIN {X 0,Y 400.074,Z 177.2,A -85,B 0,C 180,E1 -11226.718,E2 -11226.718} C_VEL
LIN {X 0,Y 398.926,Z 192.661,A -85,B 0,C 180,E1 -11230.075,E2 -11230.075} C_VEL
LIN {X 0,Y 399.244,Z 195.198,A -85,B 0,C 180,E1 -11230.208,E2 -11230.208} C_VEL
LIN {X 0,Y 403.21,Z 220.012,A -85,B 0,C 180,E1 -11230.867,E2 -11230.867} C_VEL
LIN {X 0,Y 402.021,Z 300.764,A -85,B 0,C 180,E1 -11232.382,E2 -11232.382} C_VEL
LIN {X 0,Y 401.463,Z 314.62,A -85,B 0,C 180,E1 -11232.85,E2 -11232.85} C_VEL
LIN {X 0,Y 400.812,Z 326.544,A -85,B 0,C 180,E1 -11233.444,E2 -11233.444} C_VEL
LIN {X 0,Y 400.11,Z 337.859,A -85,B 0,C 180,E1 -11234.2,E2 -11234.2} C_VEL
LIN {X 0,Y 399.313,Z 349.559,A -85,B 0,C 180,E1 -11235.214,E2 -11235.214} C_VEL
LIN {X 0,Y 398.517,Z 360.265,A -85,B 0,C 180,E1 -11236.379,E2 -11236.379} C_VEL
LIN {X 0,Y 397.882,Z 368.678,A -85,B 0,C 180,E1 -11237.503,E2 -11237.503} C_VEL
LIN {X 0,Y 397.175,Z 376.599,A -85,B 0,C 180,E1 -11238.775,E2 -11238.775} C_VEL
LIN {X 0,Y 396.633,Z 384.325,A -85,B 0,C 180,E1 -11240.308,E2 -11240.308} C_VEL
LIN {X 0,Y 396.23,Z 390.524,A -85,B 0,C 180,E1 -11241.841,E2 -11241.841} C_VEL
LIN {X 0,Y 395.939,Z 395.436,A -85,B 0,C 180,E1 -11243.374,E2 -11243.374} C_VEL
LIN {X 0,Y 395.856,Z 399.206,A -85,B 0,C 180,E1 -11244.906,E2 -11244.906} C_VEL
LIN {X 0,Y 395.767,Z 401.147,A -85,B 0,C 180,E1 -11245.926,E2 -11245.926} C_VEL
LIN {X 0,Y 395.692,Z 402.656,A -85,B 0,C 180,E1 -11246.945,E2 -11246.945} C_VEL
LIN {X 0,Y 395.721,Z 403.711,A -85,B 0,C 180,E1 -11247.963,E2 -11247.963} C_VEL
LIN {X 0,Y 395.757,Z 404.371,A -85,B 0,C 180,E1 -11248.981,E2 -11248.981} C_VEL
LIN {X 0,Y 395.761,Z 404.64,A -85,B 0,C 180,E1 -11249.999,E2 -11249.999} C_VEL
LIN {X 0,Y 395.757,Z 404.506,A -85,B 0,C 180,E1 -11251.016,E2 -11251.016} C_VEL
LIN {X 0,Y 395.72,Z 403.935,A -85,B 0,C 180,E1 -11252.034,E2 -11252.034} C_VEL
LIN {X 0,Y 395.771,Z 401.613,A -85,B 0,C 180,E1 -11254.072,E2 -11254.072} C_VEL
LIN {X 0,Y 395.875,Z 398.739,A -85,B 0,C 180,E1 -11255.602,E2 -11255.602} C_VEL
LIN {X 0,Y 396.057,Z 394.831,A -85,B 0,C 180,E1 -11257.134,E2 -11257.134} C_VEL
LIN {X 0,Y 396.388,Z 389.79,A -85,B 0,C 180,E1 -11258.667,E2 -11258.667} C_VEL
LIN {X 0,Y 396.873,Z 383.461,A -85,B 0,C 180,E1 -11260.199,E2 -11260.199} C_VEL
LIN {X 0,Y 397.518,Z 375.537,A -85,B 0,C 180,E1 -11261.73,E2 -11261.73} C_VEL
LIN {X 0,Y 398.344,Z 367.468,A -85,B 0,C 180,E1 -11262.999,E2 -11262.999} C_VEL
LIN {X 0,Y 399.115,Z 357.636,A -85,B 0,C 180,E1 -11264.271,E2 -11264.271} C_VEL
LIN {X 0,Y 400.022,Z 346.675,A -85,B 0,C 180,E1 -11265.409,E2 -11265.409} C_VEL
LIN {X 0,Y 400.975,Z 334.19,A -85,B 0,C 180,E1 -11266.416,E2 -11266.416} C_VEL
LIN {X 0,Y 401.862,Z 321.949,A -85,B 0,C 180,E1 -11267.163,E2 -11267.163} C_VEL
LIN {X 0,Y 402.49,Z 309.095,A -85,B 0,C 180,E1 -11267.726,E2 -11267.726} C_VEL
LIN {X 0,Y 402.943,Z 295.656,A -85,B 0,C 180,E1 -11268.099,E2 -11268.099} C_VEL
LIN {X 0,Y 404.058,Z 219.313,A -85,B 0,C 180,E1 -11269.543,E2 -11269.543} C_VEL
LIN {X 0,Y 400.37,Z 197.844,A -85,B 0,C 180,E1 -11270.183,E2 -11270.183} C_VEL
LIN {X 0,Y 399.335,Z 192.469,A -85,B 0,C 180,E1 -11270.386,E2 -11270.386} C_VEL
LIN {X 0,Y 399.722,Z 186.272,A -85,B 0,C 180,E1 -11271.666,E2 -11271.666} C_VEL
LIN {X 0,Y 400.402,Z 177.71,A -85,B 0,C 180,E1 -11273.534,E2 -11273.534} C_VEL
LIN {X 0,Y 399.042,Z 169.467,A -85,B 0,C 180,E1 -11275.497,E2 -11275.497} C_VEL
LIN {X 0,Y 397.073,Z 160.632,A -85,B 0,C 180,E1 -11277.751,E2 -11277.751} C_VEL
LIN {X 0,Y 397.068,Z 160.523,A -85,B 0,C 180,E1 -11280.882,E2 -11280.882} C_VEL
LIN {X 0,Y 397.111,Z 160.52,A -85,B 0,C 180,E1 -11284.493,E2 -11284.493} C_VEL
LIN {X 0,Y 397.083,Z 160.52,A -85,B 0,C 180,E1 -11288.275,E2 -11288.275} C_VEL
LIN {X 0,Y 397.044,Z 160.526,A -85,B 0,C 180,E1 -11291.975,E2 -11291.975} C_VEL
LIN {X 0,Y 397.077,Z 160.524,A -85,B 0,C 180,E1 -11295.068,E2 -11295.068} C_VEL
LIN {X 0,Y 397.043,Z 160.527,A -85,B 0,C 180,E1 -11298.022,E2 -11298.022} C_VEL
LIN {X 0,Y 397.081,Z 160.519,A -85,B 0,C 180,E1 -11301.722,E2 -11301.722} C_VEL
LIN {X 0,Y 397.107,Z 160.515,A -85,B 0,C 180,E1 -11305.504,E2 -11305.504} C_VEL
LIN {X 0,Y 397.063,Z 160.521,A -85,B 0,C 180,E1 -11309.116,E2 -11309.116} C_VEL
LIN {X 0,Y 397.05,Z 160.522,A -85,B 0,C 180,E1 -11312.251,E2 -11312.251} C_VEL
LIN {X 0,Y 397.091,Z 160.524,A -85,B 0,C 180,E1 -11314.864,E2 -11314.864} C_VEL
LIN {X 0,Y 397.083,Z 160.519,A -85,B 0,C 180,E1 -11318.18,E2 -11318.18} C_VEL
LIN {X 0,Y 397.145,Z 160.511,A -85,B 0,C 180,E1 -11321.425,E2 -11321.425} C_VEL
LIN {X 0,Y 397.164,Z 160.507,A -85,B 0,C 180,E1 -11324.607,E2 -11324.607} C_VEL
LIN {X 0,Y 397.205,Z 160.503,A -85,B 0,C 180,E1 -11327.741,E2 -11327.741} C_VEL
LIN {X 0,Y 397.222,Z 160.507,A -85,B 0,C 180,E1 -11330.837,E2 -11330.837} C_VEL
LIN {X 0,Y 397.334,Z 160.487,A -85,B 0,C 180,E1 -11333.907,E2 -11333.907} C_VEL
LIN {X 0,Y 397.43,Z 160.477,A -85,B 0,C 180,E1 -11337.973,E2 -11337.973} C_VEL
LIN {X 0,Y 397.426,Z 160.48,A -85,B 0,C 180,E1 -11342.026,E2 -11342.026} C_VEL
LIN {X 0,Y 397.308,Z 160.492,A -85,B 0,C 180,E1 -11346.686,E2 -11346.686} C_VEL
LIN {X 0,Y 397.216,Z 160.502,A -85,B 0,C 180,E1 -11349.162,E2 -11349.162} C_VEL
LIN {X 0,Y 397.2,Z 160.508,A -85,B 0,C 180,E1 -11352.258,E2 -11352.258} C_VEL
LIN {X 0,Y 397.164,Z 160.511,A -85,B 0,C 180,E1 -11355.392,E2 -11355.392} C_VEL
LIN {X 0,Y 397.143,Z 160.518,A -85,B 0,C 180,E1 -11358.574,E2 -11358.574} C_VEL
LIN {X 0,Y 397.081,Z 160.525,A -85,B 0,C 180,E1 -11361.819,E2 -11361.819} C_VEL
LIN {X 0,Y 397.089,Z 160.518,A -85,B 0,C 180,E1 -11365.136,E2 -11365.136} C_VEL
LIN {X 0,Y 397.142,Z 160.712,A -85,B 0,C 180,E1 -11368.686,E2 -11368.686} C_VEL
LIN {X 0,Y 399.272,Z 170.875,A -85,B 0,C 180,E1 -11371.282,E2 -11371.282} C_VEL
LIN {X 0,Y 399.931,Z 175.886,A -85,B 0,C 180,E1 -11372.491,E2 -11372.491} C_VEL
LIN {X 0,Y 399.633,Z 181.372,A -85,B 0,C 180,E1 -11373.677,E2 -11373.677} C_VEL
LIN {X 0,Y 403.227,Z 198.958,A -85,B 0,C 180,E1 -11374.276,E2 -11374.276} C_VEL
LIN {X 0,Y 404.319,Z 205.693,A -85,B 0,C 180,E1 -11374.472,E2 -11374.472} C_VEL
LIN {X 0,Y 402.867,Z 289.324,A -85,B 0,C 180,E1 -11376.069,E2 -11376.069} C_VEL
LIN {X 0,Y 402.416,Z 302.459,A -85,B 0,C 180,E1 -11376.521,E2 -11376.521} C_VEL
LIN {X 0,Y 401.786,Z 314.884,A -85,B 0,C 180,E1 -11377.147,E2 -11377.147} C_VEL
LIN {X 0,Y 401.045,Z 326.615,A -85,B 0,C 180,E1 -11377.949,E2 -11377.949} C_VEL
LIN {X 0,Y 400.082,Z 338.412,A -85,B 0,C 180,E1 -11378.988,E2 -11378.988} C_VEL
LIN {X 0,Y 399.128,Z 349.329,A -85,B 0,C 180,E1 -11380.206,E2 -11380.206} C_VEL
LIN {X 0,Y 398.237,Z 359.229,A -85,B 0,C 180,E1 -11381.6,E2 -11381.6} C_VEL
LIN {X 0,Y 397.623,Z 366.333,A -85,B 0,C 180,E1 -11382.821,E2 -11382.821} C_VEL
LIN {X 0,Y 396.927,Z 373.246,A -85,B 0,C 180,E1 -11384.256,E2 -11384.256} C_VEL
LIN {X 0,Y 396.508,Z 378.832,A -85,B 0,C 180,E1 -11385.691,E2 -11385.691} C_VEL
LIN {X 0,Y 396.173,Z 383.318,A -85,B 0,C 180,E1 -11387.126,E2 -11387.126} C_VEL
LIN {X 0,Y 395.918,Z 387.631,A -85,B 0,C 180,E1 -11388.947,E2 -11388.947} C_VEL
LIN {X 0,Y 395.694,Z 389.815,A -85,B 0,C 180,E1 -11390.255,E2 -11390.255} C_VEL
LIN {X 0,Y 395.59,Z 391.329,A -85,B 0,C 180,E1 -11391.554,E2 -11391.554} C_VEL
LIN {X 0,Y 395.497,Z 392.257,A -85,B 0,C 180,E1 -11393.096,E2 -11393.096} C_VEL
LIN {X 0,Y 395.491,Z 392.183,A -85,B 0,C 180,E1 -11394.828,E2 -11394.828} C_VEL
LIN {X 0,Y 395.58,Z 390.881,A -85,B 0,C 180,E1 -11396.617,E2 -11396.617} C_VEL
LIN {X 0,Y 395.793,Z 388.213,A -85,B 0,C 180,E1 -11398.464,E2 -11398.464} C_VEL
LIN {X 0,Y 396.04,Z 384.386,A -85,B 0,C 180,E1 -11400.208,E2 -11400.208} C_VEL
LIN {X 0,Y 396.346,Z 379.14,A -85,B 0,C 180,E1 -11401.942,E2 -11401.942} C_VEL
LIN {X 0,Y 396.823,Z 372.082,A -85,B 0,C 180,E1 -11403.721,E2 -11403.721} C_VEL
LIN {X 0,Y 397.379,Z 364.87,A -85,B 0,C 180,E1 -11405.165,E2 -11405.165} C_VEL
LIN {X 0,Y 398.088,Z 355.709,A -85,B 0,C 180,E1 -11406.638,E2 -11406.638} C_VEL
LIN {X 0,Y 398.898,Z 346.155,A -85,B 0,C 180,E1 -11407.878,E2 -11407.878} C_VEL
LIN {X 0,Y 399.743,Z 335.301,A -85,B 0,C 180,E1 -11409.018,E2 -11409.018} C_VEL
LIN {X 0,Y 400.495,Z 323.483,A -85,B 0,C 180,E1 -11409.991,E2 -11409.991} C_VEL
LIN {X 0,Y 401.175,Z 311.237,A -85,B 0,C 180,E1 -11410.764,E2 -11410.764} C_VEL
LIN {X 0,Y 401.741,Z 298.957,A -85,B 0,C 180,E1 -11411.33,E2 -11411.33} C_VEL
LIN {X 0,Y 402.144,Z 286.767,A -85,B 0,C 180,E1 -11411.699,E2 -11411.699} C_VEL
LIN {X 0,Y 403.228,Z 203.892,A -85,B 0,C 180,E1 -11413.255,E2 -11413.255} C_VEL
LIN {X 0,Y 399.114,Z 181.602,A -85,B 0,C 180,E1 -11413.9,E2 -11413.9} C_VEL
LIN {X 0,Y 399.196,Z 178.98,A -85,B 0,C 180,E1 -11414.427,E2 -11414.427} C_VEL
LIN {X 0,Y 399.472,Z 173.417,A -85,B 0,C 180,E1 -11415.742,E2 -11415.742} C_VEL
LIN {X 0,Y 398.623,Z 167.948,A -85,B 0,C 180,E1 -11417.11,E2 -11417.11} C_VEL
LIN {X 0,Y 397.595,Z 166.18,A -85,B 0,C 180,E1 -11417.601,E2 -11417.601} C_VEL
LIN {X 0,Y 391.194,Z 162.03,A -85,B 0,C 180,E1 -11419.121,E2 -11419.121} C_VEL
LIN {X 0,Y 390.196,Z 161.399,A -85,B 0,C 180,E1 -11419.682,E2 -11419.682} C_VEL
LIN {X 0,Y 390.169,Z 161.383,A -85,B 0,C 180,E1 -11419.78,E2 -11419.78} C_VEL
LIN {X 0,Y 390.303,Z 161.363,A -85,B 0,C 180,E1 -11422.76,E2 -11422.76} C_VEL
LIN {X 0,Y 390.223,Z 161.373,A -85,B 0,C 180,E1 -11424.835,E2 -11424.835} C_VEL
LIN {X 0,Y 390.415,Z 161.355,A -85,B 0,C 180,E1 -11427.938,E2 -11427.938} C_VEL
LIN {X 0,Y 390.546,Z 161.337,A -85,B 0,C 180,E1 -11430.001,E2 -11430.001} C_VEL
LIN {X 0,Y 390.308,Z 161.364,A -85,B 0,C 180,E1 -11433.098,E2 -11433.098} C_VEL
LIN {X 0,Y 390.315,Z 161.363,A -85,B 0,C 180,E1 -11436.203,E2 -11436.203} C_VEL
LIN {X 0,Y 390.192,Z 161.382,A -85,B 0,C 180,E1 -11439.33,E2 -11439.33} C_VEL
LIN {X 0,Y 390.17,Z 161.38,A -85,B 0,C 180,E1 -11442.484,E2 -11442.484} C_VEL
LIN {X 0,Y 390.138,Z 161.388,A -85,B 0,C 180,E1 -11445.678,E2 -11445.678} C_VEL
LIN {X 0,Y 390.101,Z 161.391,A -85,B 0,C 180,E1 -11448.923,E2 -11448.923} C_VEL
LIN {X 0,Y 390.039,Z 161.396,A -85,B 0,C 180,E1 -11452.235,E2 -11452.235} C_VEL
LIN {X 0,Y 390.118,Z 161.388,A -85,B 0,C 180,E1 -11455.744,E2 -11455.744} C_VEL
LIN {X 0,Y 390.058,Z 161.401,A -85,B 0,C 180,E1 -11459.11,E2 -11459.11} C_VEL
LIN {X 0,Y 390.042,Z 161.399,A -85,B 0,C 180,E1 -11462.722,E2 -11462.722} C_VEL
LIN {X 0,Y 390.055,Z 161.394,A -85,B 0,C 180,E1 -11465.826,E2 -11465.826} C_VEL
LIN {X 0,Y 390.067,Z 161.396,A -85,B 0,C 180,E1 -11469.219,E2 -11469.219} C_VEL
LIN {X 0,Y 390.041,Z 161.398,A -85,B 0,C 180,E1 -11472.375,E2 -11472.375} C_VEL
LIN {X 0,Y 390.043,Z 161.397,A -85,B 0,C 180,E1 -11475.355,E2 -11475.355} C_VEL
LIN {X 0,Y 390.023,Z 161.4,A -85,B 0,C 180,E1 -11478.186,E2 -11478.186} C_VEL
LIN {X 0,Y 390.062,Z 161.397,A -85,B 0,C 180,E1 -11480.905,E2 -11480.905} C_VEL
LIN {X 0,Y 390.084,Z 161.395,A -85,B 0,C 180,E1 -11484.794,E2 -11484.794} C_VEL
LIN {X 0,Y 390.024,Z 161.405,A -85,B 0,C 180,E1 -11488.496,E2 -11488.496} C_VEL
LIN {X 0,Y 390.038,Z 161.4,A -85,B 0,C 180,E1 -11492.064,E2 -11492.064} C_VEL
LIN {X 0,Y 390.063,Z 161.394,A -85,B 0,C 180,E1 -11495.519,E2 -11495.519} C_VEL
LIN {X 0,Y 390.056,Z 161.395,A -85,B 0,C 180,E1 -11498.878,E2 -11498.878} C_VEL
LIN {X 0,Y 390.128,Z 161.392,A -85,B 0,C 180,E1 -11502.167,E2 -11502.167} C_VEL
LIN {X 0,Y 390.144,Z 161.384,A -85,B 0,C 180,E1 -11505.393,E2 -11505.393} C_VEL
LIN {X 0,Y 390.146,Z 161.384,A -85,B 0,C 180,E1 -11508.572,E2 -11508.572} C_VEL
LIN {X 0,Y 390.257,Z 161.374,A -85,B 0,C 180,E1 -11512.087,E2 -11512.087} C_VEL
LIN {X 0,Y 390.204,Z 161.376,A -85,B 0,C 180,E1 -11514.834,E2 -11514.834} C_VEL
LIN {X 0,Y 390.407,Z 161.356,A -85,B 0,C 180,E1 -11517.937,E2 -11517.937} C_VEL
LIN {X 0,Y 390.411,Z 161.353,A -85,B 0,C 180,E1 -11522.064,E2 -11522.064} C_VEL
LIN {X 0,Y 390.273,Z 161.369,A -85,B 0,C 180,E1 -11526.203,E2 -11526.203} C_VEL
LIN {X 0,Y 390.189,Z 161.382,A -85,B 0,C 180,E1 -11529.33,E2 -11529.33} C_VEL
LIN {X 0,Y 390.172,Z 161.38,A -85,B 0,C 180,E1 -11532.484,E2 -11532.484} C_VEL
LIN {X 0,Y 390.138,Z 161.388,A -85,B 0,C 180,E1 -11535.677,E2 -11535.677} C_VEL
LIN {X 0,Y 390.098,Z 161.391,A -85,B 0,C 180,E1 -11538.923,E2 -11538.923} C_VEL
LIN {X 0,Y 390.036,Z 161.397,A -85,B 0,C 180,E1 -11542.235,E2 -11542.235} C_VEL
LIN {X 0,Y 390.053,Z 161.396,A -85,B 0,C 180,E1 -11545.722,E2 -11545.722} C_VEL
LIN {X 0,Y 390.024,Z 161.405,A -85,B 0,C 180,E1 -11549.113,E2 -11549.113} C_VEL
LIN {X 0,Y 390.04,Z 161.399,A -85,B 0,C 180,E1 -11552.722,E2 -11552.722} C_VEL
LIN {X 0,Y 390.043,Z 161.396,A -85,B 0,C 180,E1 -11555.822,E2 -11555.822} C_VEL
LIN {X 0,Y 390.036,Z 161.4,A -85,B 0,C 180,E1 -11559.212,E2 -11559.212} C_VEL
LIN {X 0,Y 390.031,Z 161.399,A -85,B 0,C 180,E1 -11562.372,E2 -11562.372} C_VEL
LIN {X 0,Y 390.043,Z 161.397,A -85,B 0,C 180,E1 -11565.354,E2 -11565.354} C_VEL
LIN {X 0,Y 390.017,Z 161.4,A -85,B 0,C 180,E1 -11568.184,E2 -11568.184} C_VEL
LIN {X 0,Y 390.055,Z 161.399,A -85,B 0,C 180,E1 -11570.903,E2 -11570.903} C_VEL
LIN {X 0,Y 390.055,Z 161.399,A -85,B 0,C 180,E1 -11574.789,E2 -11574.789} C_VEL
LIN {X 0,Y 390.018,Z 161.406,A -85,B 0,C 180,E1 -11578.494,E2 -11578.494} C_VEL
LIN {X 0,Y 390.025,Z 161.404,A -85,B 0,C 180,E1 -11580.887,E2 -11580.887} C_VEL
LIN {X 0,Y 390.069,Z 161.628,A -85,B 0,C 180,E1 -11582.503,E2 -11582.503} C_VEL
LIN {X 0,Y 392.428,Z 173.262,A -85,B 0,C 180,E1 -11585.393,E2 -11585.393} C_VEL
LIN {X 0,Y 393.129,Z 178.253,A -85,B 0,C 180,E1 -11586.577,E2 -11586.577} C_VEL
LIN {X 0,Y 392.031,Z 192.769,A -85,B 0,C 180,E1 -11589.765,E2 -11589.765} C_VEL
LIN {X 0,Y 392.808,Z 197.916,A -85,B 0,C 180,E1 -11589.953,E2 -11589.953} C_VEL
LIN {X 0,Y 396.448,Z 220.807,A -85,B 0,C 180,E1 -11590.574,E2 -11590.574} C_VEL
LIN {X 0,Y 395.204,Z 300.643,A -85,B 0,C 180,E1 -11592.102,E2 -11592.102} C_VEL
LIN {X 0,Y 394.661,Z 313.739,A -85,B 0,C 180,E1 -11592.545,E2 -11592.545} C_VEL
LIN {X 0,Y 394.001,Z 325.859,A -85,B 0,C 180,E1 -11593.15,E2 -11593.15} C_VEL
LIN {X 0,Y 393.243,Z 337.324,A -85,B 0,C 180,E1 -11593.917,E2 -11593.917} C_VEL
LIN {X 0,Y 392.404,Z 349.112,A -85,B 0,C 180,E1 -11594.947,E2 -11594.947} C_VEL
LIN {X 0,Y 391.656,Z 359.35,A -85,B 0,C 180,E1 -11596.07,E2 -11596.07} C_VEL
LIN {X 0,Y 390.933,Z 368.343,A -85,B 0,C 180,E1 -11597.277,E2 -11597.277} C_VEL
LIN {X 0,Y 390.176,Z 376.305,A -85,B 0,C 180,E1 -11598.571,E2 -11598.571} C_VEL
LIN {X 0,Y 389.592,Z 384.076,A -85,B 0,C 180,E1 -11600.131,E2 -11600.131} C_VEL
LIN {X 0,Y 389.161,Z 390.303,A -85,B 0,C 180,E1 -11601.692,E2 -11601.692} C_VEL
LIN {X 0,Y 388.855,Z 395.239,A -85,B 0,C 180,E1 -11603.252,E2 -11603.252} C_VEL
LIN {X 0,Y 388.752,Z 399.032,A -85,B 0,C 180,E1 -11604.813,E2 -11604.813} C_VEL
LIN {X 0,Y 388.693,Z 400.985,A -85,B 0,C 180,E1 -11605.851,E2 -11605.851} C_VEL
LIN {X 0,Y 388.602,Z 402.51,A -85,B 0,C 180,E1 -11606.889,E2 -11606.889} C_VEL
LIN {X 0,Y 388.618,Z 403.578,A -85,B 0,C 180,E1 -11607.926,E2 -11607.926} C_VEL
LIN {X 0,Y 388.656,Z 404.247,A -85,B 0,C 180,E1 -11608.963,E2 -11608.963} C_VEL
LIN {X 0,Y 388.673,Z 404.525,A -85,B 0,C 180,E1 -11609.999,E2 -11609.999} C_VEL
LIN {X 0,Y 388.656,Z 404.404,A -85,B 0,C 180,E1 -11611.035,E2 -11611.035} C_VEL
LIN {X 0,Y 388.617,Z 403.845,A -85,B 0,C 180,E1 -11612.072,E2 -11612.072} C_VEL
LIN {X 0,Y 388.699,Z 401.538,A -85,B 0,C 180,E1 -11614.146,E2 -11614.146} C_VEL
LIN {X 0,Y 388.791,Z 398.394,A -85,B 0,C 180,E1 -11615.841,E2 -11615.841} C_VEL
LIN {X 0,Y 389.005,Z 394.786,A -85,B 0,C 180,E1 -11617.264,E2 -11617.264} C_VEL
LIN {X 0,Y 389.354,Z 389.761,A -85,B 0,C 180,E1 -11618.824,E2 -11618.824} C_VEL
LIN {X 0,Y 389.883,Z 383.451,A -85,B 0,C 180,E1 -11620.384,E2 -11620.384} C_VEL
LIN {X 0,Y 390.553,Z 375.555,A -85,B 0,C 180,E1 -11621.942,E2 -11621.942} C_VEL
LIN {X 0,Y 391.429,Z 367.509,A -85,B 0,C 180,E1 -11623.232,E2 -11623.232} C_VEL
LIN {X 0,Y 392.231,Z 357.713,A -85,B 0,C 180,E1 -11624.527,E2 -11624.527} C_VEL
LIN {X 0,Y 393.181,Z 346.83,A -85,B 0,C 180,E1 -11625.684,E2 -11625.684} C_VEL
LIN {X 0,Y 394.192,Z 334.439,A -85,B 0,C 180,E1 -11626.706,E2 -11626.706} C_VEL
LIN {X 0,Y 395.118,Z 322.327,A -85,B 0,C 180,E1 -11627.466,E2 -11627.466} C_VEL
LIN {X 0,Y 395.762,Z 309.8,A -85,B 0,C 180,E1 -11628.037,E2 -11628.037} C_VEL
LIN {X 0,Y 396.265,Z 296.903,A -85,B 0,C 180,E1 -11628.415,E2 -11628.415} C_VEL
LIN {X 0,Y 397.388,Z 219.655,A -85,B 0,C 180,E1 -11629.911,E2 -11629.911} C_VEL
LIN {X 0,Y 393.436,Z 197.117,A -85,B 0,C 180,E1 -11630.608,E2 -11630.608} C_VEL
LIN {X 0,Y 392.462,Z 192.234,A -85,B 0,C 180,E1 -11630.807,E2 -11630.807} C_VEL
LIN {X 0,Y 393.487,Z 178.998,A -85,B 0,C 180,E1 -11633.693,E2 -11633.693} C_VEL
LIN {X 0,Y 392.054,Z 170.61,A -85,B 0,C 180,E1 -11635.742,E2 -11635.742} C_VEL
LIN {X 0,Y 390.021,Z 161.478,A -85,B 0,C 180,E1 -11638.133,E2 -11638.133} C_VEL
LIN {X 0,Y 390.014,Z 161.402,A -85,B 0,C 180,E1 -11641.503,E2 -11641.503} C_VEL
LIN {X 0,Y 390.063,Z 161.399,A -85,B 0,C 180,E1 -11645.207,E2 -11645.207} C_VEL
LIN {X 0,Y 390.05,Z 161.4,A -85,B 0,C 180,E1 -11649.095,E2 -11649.095} C_VEL
LIN {X 0,Y 390.022,Z 161.4,A -85,B 0,C 180,E1 -11652.37,E2 -11652.37} C_VEL
LIN {X 0,Y 390.032,Z 161.405,A -85,B 0,C 180,E1 -11655.352,E2 -11655.352} C_VEL
LIN {X 0,Y 390.006,Z 161.403,A -85,B 0,C 180,E1 -11658.183,E2 -11658.183} C_VEL
LIN {X 0,Y 390.049,Z 161.4,A -85,B 0,C 180,E1 -11660.902,E2 -11660.902} C_VEL
LIN {X 0,Y 390.06,Z 161.398,A -85,B 0,C 180,E1 -11664.79,E2 -11664.79} C_VEL
LIN {X 0,Y 390.009,Z 161.402,A -85,B 0,C 180,E1 -11668.494,E2 -11668.494} C_VEL
LIN {X 0,Y 390.005,Z 161.4,A -85,B 0,C 180,E1 -11672.002,E2 -11672.002} C_VEL
LIN {X 0,Y 390.03,Z 161.398,A -85,B 0,C 180,E1 -11675.516,E2 -11675.516} C_VEL
LIN {X 0,Y 390.044,Z 161.402,A -85,B 0,C 180,E1 -11678.877,E2 -11678.877} C_VEL
LIN {X 0,Y 390.099,Z 161.388,A -85,B 0,C 180,E1 -11682.165,E2 -11682.165} C_VEL
LIN {X 0,Y 390.129,Z 161.385,A -85,B 0,C 180,E1 -11685.392,E2 -11685.392} C_VEL
LIN {X 0,Y 390.132,Z 161.384,A -85,B 0,C 180,E1 -11688.57,E2 -11688.57} C_VEL
LIN {X 0,Y 390.257,Z 161.37,A -85,B 0,C 180,E1 -11692.071,E2 -11692.071} C_VEL
LIN {X 0,Y 390.199,Z 161.381,A -85,B 0,C 180,E1 -11694.833,E2 -11694.833} C_VEL
LIN {X 0,Y 390.397,Z 161.353,A -85,B 0,C 180,E1 -11697.936,E2 -11697.936} C_VEL
LIN {X 0,Y 390.394,Z 161.356,A -85,B 0,C 180,E1 -11702.063,E2 -11702.063} C_VEL
LIN {X 0,Y 390.261,Z 161.369,A -85,B 0,C 180,E1 -11706.682,E2 -11706.682} C_VEL
LIN {X 0,Y 390.174,Z 161.379,A -85,B 0,C 180,E1 -11709.329,E2 -11709.329} C_VEL
LIN {X 0,Y 390.181,Z 161.381,A -85,B 0,C 180,E1 -11713.438,E2 -11713.438} C_VEL
LIN {X 0,Y 390.116,Z 161.39,A -85,B 0,C 180,E1 -11717.298,E2 -11717.298} C_VEL
LIN {X 0,Y 390.074,Z 161.397,A -85,B 0,C 180,E1 -11720.47,E2 -11720.47} C_VEL
LIN {X 0,Y 390.048,Z 161.399,A -85,B 0,C 180,E1 -11723.353,E2 -11723.353} C_VEL
LIN {X 0,Y 390.016,Z 161.402,A -85,B 0,C 180,E1 -11726.775,E2 -11726.775} C_VEL
LIN {X 0,Y 390.038,Z 161.498,A -85,B 0,C 180,E1 -11728.279,E2 -11728.279} C_VEL
LIN {X 0,Y 392.168,Z 171.147,A -85,B 0,C 180,E1 -11730.835,E2 -11730.835} C_VEL
LIN {X 0,Y 393.022,Z 176.378,A -85,B 0,C 180,E1 -11732.139,E2 -11732.139} C_VEL
LIN {X 0,Y 392.813,Z 181.534,A -85,B 0,C 180,E1 -11733.266,E2 -11733.266} C_VEL
LIN {X 0,Y 395.249,Z 192.847,A -85,B 0,C 180,E1 -11733.686,E2 -11733.686} C_VEL
LIN {X 0,Y 397.66,Z 205.785,A -85,B 0,C 180,E1 -11734.094,E2 -11734.094} C_VEL
LIN {X 0,Y 396.218,Z 289.114,A -85,B 0,C 180,E1 -11735.715,E2 -11735.715} C_VEL
LIN {X 0,Y 395.715,Z 302.8,A -85,B 0,C 180,E1 -11736.194,E2 -11736.194} C_VEL
LIN {X 0,Y 395.076,Z 315.045,A -85,B 0,C 180,E1 -11736.825,E2 -11736.825} C_VEL
LIN {X 0,Y 394.287,Z 326.558,A -85,B 0,C 180,E1 -11737.623,E2 -11737.623} C_VEL
LIN {X 0,Y 393.433,Z 336.819,A -85,B 0,C 180,E1 -11738.525,E2 -11738.525} C_VEL
LIN {X 0,Y 392.463,Z 347.109,A -85,B 0,C 180,E1 -11739.647,E2 -11739.647} C_VEL
LIN {X 0,Y 391.639,Z 356.069,A -85,B 0,C 180,E1 -11740.849,E2 -11740.849} C_VEL
LIN {X 0,Y 390.806,Z 364.797,A -85,B 0,C 180,E1 -11742.279,E2 -11742.279} C_VEL
LIN {X 0,Y 390.016,Z 372.618,A -85,B 0,C 180,E1 -11743.883,E2 -11743.883} C_VEL
LIN {X 0,Y 389.534,Z 378.14,A -85,B 0,C 180,E1 -11745.283,E2 -11745.283} C_VEL
LIN {X 0,Y 389.187,Z 382.6,A -85,B 0,C 180,E1 -11746.671,E2 -11746.671} C_VEL
LIN {X 0,Y 388.977,Z 386.124,A -85,B 0,C 180,E1 -11748.05,E2 -11748.05} C_VEL
LIN {X 0,Y 388.76,Z 388.758,A -85,B 0,C 180,E1 -11749.4,E2 -11749.4} C_VEL
LIN {X 0,Y 388.528,Z 391.022,A -85,B 0,C 180,E1 -11751.06,E2 -11751.06} C_VEL
LIN {X 0,Y 388.42,Z 392.247,A -85,B 0,C 180,E1 -11752.761,E2 -11752.761} C_VEL
LIN {X 0,Y 388.388,Z 392.365,A -85,B 0,C 180,E1 -11754.618,E2 -11754.618} C_VEL
LIN {X 0,Y 388.47,Z 391.321,A -85,B 0,C 180,E1 -11756.325,E2 -11756.325} C_VEL
LIN {X 0,Y 388.65,Z 388.871,A -85,B 0,C 180,E1 -11758.2,E2 -11758.2} C_VEL
LIN {X 0,Y 388.927,Z 384.825,A -85,B 0,C 180,E1 -11760.154,E2 -11760.154} C_VEL
LIN {X 0,Y 389.276,Z 379.42,A -85,B 0,C 180,E1 -11762.006,E2 -11762.006} C_VEL
LIN {X 0,Y 389.78,Z 372.53,A -85,B 0,C 180,E1 -11763.787,E2 -11763.787} C_VEL
LIN {X 0,Y 390.333,Z 365.399,A -85,B 0,C 180,E1 -11765.254,E2 -11765.254} C_VEL
LIN {X 0,Y 391.073,Z 356.644,A -85,B 0,C 180,E1 -11766.713,E2 -11766.713} C_VEL
LIN {X 0,Y 391.949,Z 346.281,A -85,B 0,C 180,E1 -11768.093,E2 -11768.093} C_VEL
LIN {X 0,Y 392.767,Z 336.266,A -85,B 0,C 180,E1 -11769.169,E2 -11769.169} C_VEL
LIN {X 0,Y 393.556,Z 324.631,A -85,B 0,C 180,E1 -11770.167,E2 -11770.167} C_VEL
LIN {X 0,Y 394.29,Z 312.526,A -85,B 0,C 180,E1 -11770.961,E2 -11770.961} C_VEL
LIN {X 0,Y 394.872,Z 299.956,A -85,B 0,C 180,E1 -11771.568,E2 -11771.568} C_VEL
LIN {X 0,Y 395.334,Z 287.048,A -85,B 0,C 180,E1 -11771.976,E2 -11771.976} C_VEL
LIN {X 0,Y 396.412,Z 204.496,A -85,B 0,C 180,E1 -11773.558,E2 -11773.558} C_VEL
LIN {X 0,Y 392.22,Z 181.796,A -85,B 0,C 180,E1 -11774.226,E2 -11774.226} C_VEL
LIN {X 0,Y 392.193,Z 180.618,A -85,B 0,C 180,E1 -11774.409,E2 -11774.409} C_VEL
LIN {X 0,Y 392.531,Z 174.97,A -85,B 0,C 180,E1 -11775.75,E2 -11775.75} C_VEL
LIN {X 0,Y 391.044,Z 165.899,A -85,B 0,C 180,E1 -11778.073,E2 -11778.073} C_VEL
LIN {X 0,Y 390.189,Z 161.472,A -85,B 0,C 180,E1 -11779.297,E2 -11779.297} C_VEL
LIN {X 0,Y 390.169,Z 161.383,A -85,B 0,C 180,E1 -11779.78,E2 -11779.78} C_VEL
LIN {X 0,Y 389.516,Z 161.464,A -85,B 0,C 180,E1 -11780.643,E2 -11780.643} C_VEL
LIN {X 0,Y 386.727,Z 161.814,A -85,B 0,C 180,E1 -11782.046,E2 -11782.046} C_VEL
LIN {X 0,Y 384.35,Z 162.109,A -85,B 0,C 180,E1 -11783.181,E2 -11783.181} C_VEL
LIN {X 0,Y 383.308,Z 162.239,A -85,B 0,C 180,E1 -11784.057,E2 -11784.057} C_VEL
LIN {X 0,Y 383.211,Z 162.247,A -85,B 0,C 180,E1 -11784.353,E2 -11784.353} C_VEL
LIN {X 0,Y 383.382,Z 162.231,A -85,B 0,C 180,E1 -11787.9,E2 -11787.9} C_VEL
LIN {X 0,Y 383.515,Z 162.213,A -85,B 0,C 180,E1 -11790.001,E2 -11790.001} C_VEL
LIN {X 0,Y 383.244,Z 162.244,A -85,B 0,C 180,E1 -11793.155,E2 -11793.155} C_VEL
LIN {X 0,Y 383.27,Z 162.24,A -85,B 0,C 180,E1 -11796.318,E2 -11796.318} C_VEL
LIN {X 0,Y 383.142,Z 162.262,A -85,B 0,C 180,E1 -11799.503,E2 -11799.503} C_VEL
LIN {X 0,Y 383.135,Z 162.257,A -85,B 0,C 180,E1 -11802.717,E2 -11802.717} C_VEL
LIN {X 0,Y 383.079,Z 162.265,A -85,B 0,C 180,E1 -11805.974,E2 -11805.974} C_VEL
LIN {X 0,Y 383.057,Z 162.272,A -85,B 0,C 180,E1 -11809.285,E2 -11809.285} C_VEL
LIN {X 0,Y 383.007,Z 162.273,A -85,B 0,C 180,E1 -11812.666,E2 -11812.666} C_VEL
LIN {X 0,Y 383.079,Z 162.263,A -85,B 0,C 180,E1 -11816.124,E2 -11816.124} C_VEL
LIN {X 0,Y 382.991,Z 162.275,A -85,B 0,C 180,E1 -11819.701,E2 -11819.701} C_VEL
LIN {X 0,Y 383.002,Z 162.275,A -85,B 0,C 180,E1 -11823.402,E2 -11823.402} C_VEL
LIN {X 0,Y 383.031,Z 162.27,A -85,B 0,C 180,E1 -11826.165,E2 -11826.165} C_VEL
LIN {X 0,Y 383.007,Z 162.272,A -85,B 0,C 180,E1 -11829.959,E2 -11829.959} C_VEL
LIN {X 0,Y 383.005,Z 162.279,A -85,B 0,C 180,E1 -11832.779,E2 -11832.779} C_VEL
LIN {X 0,Y 382.996,Z 162.274,A -85,B 0,C 180,E1 -11835.79,E2 -11835.79} C_VEL
LIN {X 0,Y 382.971,Z 162.282,A -85,B 0,C 180,E1 -11838.8,E2 -11838.8} C_VEL
LIN {X 0,Y 382.994,Z 162.275,A -85,B 0,C 180,E1 -11842.098,E2 -11842.098} C_VEL
LIN {X 0,Y 383.018,Z 162.271,A -85,B 0,C 180,E1 -11845.333,E2 -11845.333} C_VEL
LIN {X 0,Y 382.982,Z 162.276,A -85,B 0,C 180,E1 -11849.082,E2 -11849.082} C_VEL
LIN {X 0,Y 382.993,Z 162.277,A -85,B 0,C 180,E1 -11852.694,E2 -11852.694} C_VEL
LIN {X 0,Y 383.022,Z 162.276,A -85,B 0,C 180,E1 -11856.192,E2 -11856.192} C_VEL
LIN {X 0,Y 383.056,Z 162.267,A -85,B 0,C 180,E1 -11859.599,E2 -11859.599} C_VEL
LIN {X 0,Y 383.106,Z 162.26,A -85,B 0,C 180,E1 -11862.932,E2 -11862.932} C_VEL
LIN {X 0,Y 383.127,Z 162.26,A -85,B 0,C 180,E1 -11866.465,E2 -11866.465} C_VEL
LIN {X 0,Y 383.143,Z 162.257,A -85,B 0,C 180,E1 -11870.498,E2 -11870.498} C_VEL
LIN {X 0,Y 383.239,Z 162.247,A -85,B 0,C 180,E1 -11873.683,E2 -11873.683} C_VEL
LIN {X 0,Y 383.373,Z 162.233,A -85,B 0,C 180,E1 -11877.899,E2 -11877.899} C_VEL
LIN {X 0,Y 383.377,Z 162.229,A -85,B 0,C 180,E1 -11882.102,E2 -11882.102} C_VEL
LIN {X 0,Y 383.231,Z 162.245,A -85,B 0,C 180,E1 -11886.318,E2 -11886.318} C_VEL
LIN {X 0,Y 383.14,Z 162.262,A -85,B 0,C 180,E1 -11889.503,E2 -11889.503} C_VEL
LIN {X 0,Y 383.128,Z 162.263,A -85,B 0,C 180,E1 -11893.536,E2 -11893.536} C_VEL
LIN {X 0,Y 383.078,Z 162.27,A -85,B 0,C 180,E1 -11897.445,E2 -11897.445} C_VEL
LIN {X 0,Y 383.019,Z 162.271,A -85,B 0,C 180,E1 -11900.642,E2 -11900.642} C_VEL
LIN {X 0,Y 383.01,Z 162.273,A -85,B 0,C 180,E1 -11903.809,E2 -11903.809} C_VEL
LIN {X 0,Y 382.967,Z 162.283,A -85,B 0,C 180,E1 -11907.309,E2 -11907.309} C_VEL
LIN {X 0,Y 382.98,Z 162.28,A -85,B 0,C 180,E1 -11910.919,E2 -11910.919} C_VEL
LIN {X 0,Y 383.013,Z 162.274,A -85,B 0,C 180,E1 -11914.669,E2 -11914.669} C_VEL
LIN {X 0,Y 382.993,Z 162.274,A -85,B 0,C 180,E1 -11917.902,E2 -11917.902} C_VEL
LIN {X 0,Y 382.962,Z 162.28,A -85,B 0,C 180,E1 -11921.351,E2 -11921.351} C_VEL
LIN {X 0,Y 382.992,Z 162.276,A -85,B 0,C 180,E1 -11924.302,E2 -11924.302} C_VEL
LIN {X 0,Y 382.985,Z 162.277,A -85,B 0,C 180,E1 -11927.236,E2 -11927.236} C_VEL
LIN {X 0,Y 382.985,Z 162.279,A -85,B 0,C 180,E1 -11930.42,E2 -11930.42} C_VEL
LIN {X 0,Y 383.007,Z 162.274,A -85,B 0,C 180,E1 -11934.042,E2 -11934.042} C_VEL
LIN {X 0,Y 382.971,Z 162.277,A -85,B 0,C 180,E1 -11937.583,E2 -11937.583} C_VEL
LIN {X 0,Y 382.976,Z 162.282,A -85,B 0,C 180,E1 -11940.298,E2 -11940.298} C_VEL
LIN {X 0,Y 383.022,Z 162.421,A -85,B 0,C 180,E1 -11942.195,E2 -11942.195} C_VEL
LIN {X 0,Y 385.404,Z 174.214,A -85,B 0,C 180,E1 -11945.202,E2 -11945.202} C_VEL
LIN {X 0,Y 386.159,Z 179.132,A -85,B 0,C 180,E1 -11946.396,E2 -11946.396} C_VEL
LIN {X 0,Y 385.111,Z 192.764,A -85,B 0,C 180,E1 -11949.432,E2 -11949.432} C_VEL
LIN {X 0,Y 388.372,Z 212.628,A -85,B 0,C 180,E1 -11950.029,E2 -11950.029} C_VEL
LIN {X 0,Y 389.692,Z 221.372,A -85,B 0,C 180,E1 -11950.268,E2 -11950.268} C_VEL
LIN {X 0,Y 388.384,Z 300.52,A -85,B 0,C 180,E1 -11951.81,E2 -11951.81} C_VEL
LIN {X 0,Y 387.825,Z 313.613,A -85,B 0,C 180,E1 -11952.261,E2 -11952.261} C_VEL
LIN {X 0,Y 387.114,Z 326.3,A -85,B 0,C 180,E1 -11952.909,E2 -11952.909} C_VEL
LIN {X 0,Y 386.268,Z 338.416,A -85,B 0,C 180,E1 -11953.754,E2 -11953.754} C_VEL
LIN {X 0,Y 385.401,Z 349.969,A -85,B 0,C 180,E1 -11954.802,E2 -11954.802} C_VEL
LIN {X 0,Y 384.553,Z 360.941,A -85,B 0,C 180,E1 -11956.057,E2 -11956.057} C_VEL
LIN {X 0,Y 383.82,Z 369.737,A -85,B 0,C 180,E1 -11957.306,E2 -11957.306} C_VEL
LIN {X 0,Y 382.941,Z 378.792,A -85,B 0,C 180,E1 -11958.888,E2 -11958.888} C_VEL
LIN {X 0,Y 382.392,Z 386.084,A -85,B 0,C 180,E1 -11960.478,E2 -11960.478} C_VEL
LIN {X 0,Y 381.992,Z 391.897,A -85,B 0,C 180,E1 -11962.068,E2 -11962.068} C_VEL
LIN {X 0,Y 381.694,Z 396.975,A -85,B 0,C 180,E1 -11963.874,E2 -11963.874} C_VEL
LIN {X 0,Y 381.62,Z 400.823,A -85,B 0,C 180,E1 -11965.774,E2 -11965.774} C_VEL
LIN {X 0,Y 381.516,Z 402.363,A -85,B 0,C 180,E1 -11966.831,E2 -11966.831} C_VEL
LIN {X 0,Y 381.516,Z 403.445,A -85,B 0,C 180,E1 -11967.888,E2 -11967.888} C_VEL
LIN {X 0,Y 381.555,Z 404.123,A -85,B 0,C 180,E1 -11968.944,E2 -11968.944} C_VEL
LIN {X 0,Y 381.588,Z 404.41,A -85,B 0,C 180,E1 -11969.999,E2 -11969.999} C_VEL
LIN {X 0,Y 381.554,Z 404.301,A -85,B 0,C 180,E1 -11971.054,E2 -11971.054} C_VEL
LIN {X 0,Y 381.515,Z 403.754,A -85,B 0,C 180,E1 -11972.11,E2 -11972.11} C_VEL
LIN {X 0,Y 381.629,Z 401.462,A -85,B 0,C 180,E1 -11974.223,E2 -11974.223} C_VEL
LIN {X 0,Y 381.699,Z 399.698,A -85,B 0,C 180,E1 -11975.281,E2 -11975.281} C_VEL
LIN {X 0,Y 381.844,Z 396.178,A -85,B 0,C 180,E1 -11976.87,E2 -11976.87} C_VEL
LIN {X 0,Y 382.161,Z 391.558,A -85,B 0,C 180,E1 -11978.459,E2 -11978.459} C_VEL
LIN {X 0,Y 382.752,Z 384.575,A -85,B 0,C 180,E1 -11980.312,E2 -11980.312} C_VEL
LIN {X 0,Y 383.472,Z 377.029,A -85,B 0,C 180,E1 -11981.897,E2 -11981.897} C_VEL
LIN {X 0,Y 384.317,Z 369.335,A -85,B 0,C 180,E1 -11983.213,E2 -11983.213} C_VEL
LIN {X 0,Y 385.187,Z 359.526,A -85,B 0,C 180,E1 -11984.587,E2 -11984.587} C_VEL
LIN {X 0,Y 386.236,Z 348.326,A -85,B 0,C 180,E1 -11985.838,E2 -11985.838} C_VEL
LIN {X 0,Y 387.266,Z 336.491,A -85,B 0,C 180,E1 -11986.878,E2 -11986.878} C_VEL
LIN {X 0,Y 388.281,Z 323.852,A -85,B 0,C 180,E1 -11987.715,E2 -11987.715} C_VEL
LIN {X 0,Y 389.046,Z 310.512,A -85,B 0,C 180,E1 -11988.36,E2 -11988.36} C_VEL
LIN {X 0,Y 389.599,Z 296.715,A -85,B 0,C 180,E1 -11988.775,E2 -11988.775} C_VEL
LIN {X 0,Y 390.812,Z 220.625,A -85,B 0,C 180,E1 -11990.275,E2 -11990.275} C_VEL
LIN {X 0,Y 386.839,Z 197.969,A -85,B 0,C 180,E1 -11990.994,E2 -11990.994} C_VEL
LIN {X 0,Y 385.659,Z 192.178,A -85,B 0,C 180,E1 -11991.227,E2 -11991.227} C_VEL
LIN {X 0,Y 386.582,Z 181.534,A -85,B 0,C 180,E1 -11993.574,E2 -11993.574} C_VEL
LIN {X 0,Y 385.843,Z 175.466,A -85,B 0,C 180,E1 -11995.054,E2 -11995.054} C_VEL
LIN {X 0,Y 383.488,Z 164.648,A -85,B 0,C 180,E1 -11997.84,E2 -11997.84} C_VEL
LIN {X 0,Y 382.983,Z 162.317,A -85,B 0,C 180,E1 -11998.533,E2 -11998.533} C_VEL
LIN {X 0,Y 383.001,Z 162.278,A -85,B 0,C 180,E1 -12002.149,E2 -12002.149} C_VEL
LIN {X 0,Y 383.006,Z 162.277,A -85,B 0,C 180,E1 -12004.667,E2 -12004.667} C_VEL
LIN {X 0,Y 382.986,Z 162.278,A -85,B 0,C 180,E1 -12007.9,E2 -12007.9} C_VEL
LIN {X 0,Y 382.954,Z 162.285,A -85,B 0,C 180,E1 -12011.349,E2 -12011.349} C_VEL
LIN {X 0,Y 382.981,Z 162.276,A -85,B 0,C 180,E1 -12014.3,E2 -12014.3} C_VEL
LIN {X 0,Y 382.974,Z 162.28,A -85,B 0,C 180,E1 -12017.235,E2 -12017.235} C_VEL
LIN {X 0,Y 382.977,Z 162.278,A -85,B 0,C 180,E1 -12020.418,E2 -12020.418} C_VEL
LIN {X 0,Y 383.005,Z 162.275,A -85,B 0,C 180,E1 -12024.042,E2 -12024.042} C_VEL
LIN {X 0,Y 382.973,Z 162.279,A -85,B 0,C 180,E1 -12027.578,E2 -12027.578} C_VEL
LIN {X 0,Y 382.964,Z 162.278,A -85,B 0,C 180,E1 -12030.297,E2 -12030.297} C_VEL
LIN {X 0,Y 382.992,Z 162.275,A -85,B 0,C 180,E1 -12034.044,E2 -12034.044} C_VEL
LIN {X 0,Y 382.975,Z 162.276,A -85,B 0,C 180,E1 -12037.333,E2 -12037.333} C_VEL
LIN {X 0,Y 383.047,Z 162.265,A -85,B 0,C 180,E1 -12040.715,E2 -12040.715} C_VEL
LIN {X 0,Y 383.067,Z 162.264,A -85,B 0,C 180,E1 -12044.026,E2 -12044.026} C_VEL
LIN {X 0,Y 383.124,Z 162.259,A -85,B 0,C 180,E1 -12047.283,E2 -12047.283} C_VEL
LIN {X 0,Y 383.129,Z 162.26,A -85,B 0,C 180,E1 -12050.497,E2 -12050.497} C_VEL
LIN {X 0,Y 383.247,Z 162.242,A -85,B 0,C 180,E1 -12053.683,E2 -12053.683} C_VEL
LIN {X 0,Y 383.363,Z 162.229,A -85,B 0,C 180,E1 -12057.898,E2 -12057.898} C_VEL
LIN {X 0,Y 383.36,Z 162.232,A -85,B 0,C 180,E1 -12062.101,E2 -12062.101} C_VEL
LIN {X 0,Y 383.22,Z 162.246,A -85,B 0,C 180,E1 -12066.674,E2 -12066.674} C_VEL
LIN {X 0,Y 383.124,Z 162.258,A -85,B 0,C 180,E1 -12069.502,E2 -12069.502} C_VEL
LIN {X 0,Y 383.112,Z 162.262,A -85,B 0,C 180,E1 -12073.536,E2 -12073.536} C_VEL
LIN {X 0,Y 383.08,Z 162.267,A -85,B 0,C 180,E1 -12077.069,E2 -12077.069} C_VEL
LIN {X 0,Y 383.015,Z 162.275,A -85,B 0,C 180,E1 -12080.647,E2 -12080.647} C_VEL
LIN {X 0,Y 382.996,Z 162.279,A -85,B 0,C 180,E1 -12083.809,E2 -12083.809} C_VEL
LIN {X 0,Y 382.957,Z 162.282,A -85,B 0,C 180,E1 -12087.309,E2 -12087.309} C_VEL
LIN {X 0,Y 382.98,Z 162.409,A -85,B 0,C 180,E1 -12087.922,E2 -12087.922} C_VEL
LIN {X 0,Y 385.296,Z 172.754,A -85,B 0,C 180,E1 -12090.712,E2 -12090.712} C_VEL
LIN {X 0,Y 386.134,Z 178.508,A -85,B 0,C 180,E1 -12092.166,E2 -12092.166} C_VEL
LIN {X 0,Y 385.989,Z 181.682,A -85,B 0,C 180,E1 -12092.838,E2 -12092.838} C_VEL
LIN {X 0,Y 388.556,Z 193.273,A -85,B 0,C 180,E1 -12093.287,E2 -12093.287} C_VEL
LIN {X 0,Y 391.15,Z 207.756,A -85,B 0,C 180,E1 -12093.751,E2 -12093.751} C_VEL
LIN {X 0,Y 389.548,Z 289.796,A -85,B 0,C 180,E1 -12095.376,E2 -12095.376} C_VEL
LIN {X 0,Y 389.034,Z 303.156,A -85,B 0,C 180,E1 -12095.856,E2 -12095.856} C_VEL
LIN {X 0,Y 388.325,Z 315.68,A -85,B 0,C 180,E1 -12096.517,E2 -12096.517} C_VEL
LIN {X 0,Y 387.435,Z 327.875,A -85,B 0,C 180,E1 -12097.396,E2 -12097.396} C_VEL
LIN {X 0,Y 386.466,Z 338.779,A -85,B 0,C 180,E1 -12098.401,E2 -12098.401} C_VEL
LIN {X 0,Y 385.396,Z 349.666,A -85,B 0,C 180,E1 -12099.661,E2 -12099.661} C_VEL
LIN {X 0,Y 384.532,Z 358.499,A -85,B 0,C 180,E1 -12100.935,E2 -12100.935} C_VEL
LIN {X 0,Y 383.677,Z 366.954,A -85,B 0,C 180,E1 -12102.431,E2 -12102.431} C_VEL
LIN {X 0,Y 382.932,Z 373.795,A -85,B 0,C 180,E1 -12103.919,E2 -12103.919} C_VEL
LIN {X 0,Y 382.363,Z 380.288,A -85,B 0,C 180,E1 -12105.699,E2 -12105.699} C_VEL
LIN {X 0,Y 381.98,Z 385.004,A -85,B 0,C 180,E1 -12107.387,E2 -12107.387} C_VEL
LIN {X 0,Y 381.71,Z 388.411,A -85,B 0,C 180,E1 -12109.015,E2 -12109.015} C_VEL
LIN {X 0,Y 381.468,Z 390.834,A -85,B 0,C 180,E1 -12110.695,E2 -12110.695} C_VEL
LIN {X 0,Y 381.327,Z 392.284,A -85,B 0,C 180,E1 -12112.542,E2 -12112.542} C_VEL
LIN {X 0,Y 381.298,Z 392.542,A -85,B 0,C 180,E1 -12114.193,E2 -12114.193} C_VEL
LIN {X 0,Y 381.363,Z 391.678,A -85,B 0,C 180,E1 -12116.025,E2 -12116.025} C_VEL
LIN {X 0,Y 381.525,Z 389.501,A -85,B 0,C 180,E1 -12117.924,E2 -12117.924} C_VEL
LIN {X 0,Y 381.678,Z 387.713,A -85,B 0,C 180,E1 -12118.966,E2 -12118.966} C_VEL
LIN {X 0,Y 381.937,Z 383.433,A -85,B 0,C 180,E1 -12120.817,E2 -12120.817} C_VEL
LIN {X 0,Y 382.353,Z 377.722,A -85,B 0,C 180,E1 -12122.645,E2 -12122.645} C_VEL
LIN {X 0,Y 382.891,Z 370.837,A -85,B 0,C 180,E1 -12124.345,E2 -12124.345} C_VEL
LIN {X 0,Y 383.602,Z 362.652,A -85,B 0,C 180,E1 -12125.945,E2 -12125.945} C_VEL
LIN {X 0,Y 384.419,Z 353.26,A -85,B 0,C 180,E1 -12127.425,E2 -12127.425} C_VEL
LIN {X 0,Y 385.329,Z 342.691,A -85,B 0,C 180,E1 -12128.748,E2 -12128.748} C_VEL
LIN {X 0,Y 386.281,Z 331.017,A -85,B 0,C 180,E1 -12129.911,E2 -12129.911} C_VEL
LIN {X 0,Y 387,Z 319.743,A -85,B 0,C 180,E1 -12130.79,E2 -12130.79} C_VEL
LIN {X 0,Y 387.661,Z 307.696,A -85,B 0,C 180,E1 -12131.504,E2 -12131.504} C_VEL
LIN {X 0,Y 388.274,Z 294.34,A -85,B 0,C 180,E1 -12132.063,E2 -12132.063} C_VEL
LIN {X 0,Y 388.615,Z 280.845,A -85,B 0,C 180,E1 -12132.403,E2 -12132.403} C_VEL
LIN {X 0,Y 389.779,Z 206.127,A -85,B 0,C 180,E1 -12133.84,E2 -12133.84} C_VEL
LIN {X 0,Y 385.361,Z 182.218,A -85,B 0,C 180,E1 -12134.556,E2 -12134.556} C_VEL
LIN {X 0,Y 385.268,Z 181.157,A -85,B 0,C 180,E1 -12134.664,E2 -12134.664} C_VEL
LIN {X 0,Y 385.53,Z 175.468,A -85,B 0,C 180,E1 -12136.024,E2 -12136.024} C_VEL
LIN {X 0,Y 383.562,Z 164.504,A -85,B 0,C 180,E1 -12138.909,E2 -12138.909} C_VEL
LIN {X 0,Y 383.153,Z 162.316,A -85,B 0,C 180,E1 -12139.566,E2 -12139.566} C_VEL
LIN {X 0,Y 383.255,Z 162.242,A -85,B 0,C 180,E1 -12142.626,E2 -12142.626} C_VEL
LIN {X 0,Y 383.211,Z 162.247,A -85,B 0,C 180,E1 -12144.353,E2 -12144.353} C_VEL
LIN {X 0,Y 382.506,Z 162.337,A -85,B 0,C 180,E1 -12145.231,E2 -12145.231} C_VEL
LIN {X 0,Y 379.638,Z 162.693,A -85,B 0,C 180,E1 -12146.658,E2 -12146.658} C_VEL
LIN {X 0,Y 377.279,Z 162.992,A -85,B 0,C 180,E1 -12147.811,E2 -12147.811} C_VEL
LIN {X 0,Y 376.333,Z 163.105,A -85,B 0,C 180,E1 -12148.703,E2 -12148.703} C_VEL
LIN {X 0,Y 376.291,Z 163.109,A -85,B 0,C 180,E1 -12149.005,E2 -12149.005} C_VEL
LIN {X 0,Y 376.484,Z 163.089,A -85,B 0,C 180,E1 -12150.001,E2 -12150.001} C_VEL
LIN {X 0,Y 376.182,Z 163.124,A -85,B 0,C 180,E1 -12153.214,E2 -12153.214} C_VEL
LIN {X 0,Y 376.227,Z 163.117,A -85,B 0,C 180,E1 -12156.436,E2 -12156.436} C_VEL
LIN {X 0,Y 376.112,Z 163.136,A -85,B 0,C 180,E1 -12159.683,E2 -12159.683} C_VEL
LIN {X 0,Y 376.088,Z 163.138,A -85,B 0,C 180,E1 -12163.659,E2 -12163.659} C_VEL
LIN {X 0,Y 376.042,Z 163.144,A -85,B 0,C 180,E1 -12167.608,E2 -12167.608} C_VEL
LIN {X 0,Y 375.977,Z 163.15,A -85,B 0,C 180,E1 -12170.833,E2 -12170.833} C_VEL
LIN {X 0,Y 375.993,Z 163.146,A -85,B 0,C 180,E1 -12174.282,E2 -12174.282} C_VEL
LIN {X 0,Y 376.019,Z 163.144,A -85,B 0,C 180,E1 -12176.653,E2 -12176.653} C_VEL
LIN {X 0,Y 375.964,Z 163.15,A -85,B 0,C 180,E1 -12180.313,E2 -12180.313} C_VEL
LIN {X 0,Y 375.959,Z 163.15,A -85,B 0,C 180,E1 -12184.112,E2 -12184.112} C_VEL
LIN {X 0,Y 375.952,Z 163.155,A -85,B 0,C 180,E1 -12186.742,E2 -12186.742} C_VEL
LIN {X 0,Y 375.987,Z 163.147,A -85,B 0,C 180,E1 -12189.971,E2 -12189.971} C_VEL
LIN {X 0,Y 375.929,Z 163.154,A -85,B 0,C 180,E1 -12193.767,E2 -12193.767} C_VEL
LIN {X 0,Y 375.934,Z 163.159,A -85,B 0,C 180,E1 -12196.811,E2 -12196.811} C_VEL
LIN {X 0,Y 375.941,Z 163.158,A -85,B 0,C 180,E1 -12200.535,E2 -12200.535} C_VEL
LIN {X 0,Y 375.963,Z 163.15,A -85,B 0,C 180,E1 -12203.497,E2 -12203.497} C_VEL
LIN {X 0,Y 375.96,Z 163.151,A -85,B 0,C 180,E1 -12205.889,E2 -12205.889} C_VEL
LIN {X 0,Y 375.962,Z 163.15,A -85,B 0,C 180,E1 -12209.688,E2 -12209.688} C_VEL
LIN {X 0,Y 375.933,Z 163.153,A -85,B 0,C 180,E1 -12213.342,E2 -12213.342} C_VEL
LIN {X 0,Y 375.984,Z 163.148,A -85,B 0,C 180,E1 -12216.888,E2 -12216.888} C_VEL
LIN {X 0,Y 375.998,Z 163.151,A -85,B 0,C 180,E1 -12220.34,E2 -12220.34} C_VEL
LIN {X 0,Y 376.029,Z 163.144,A -85,B 0,C 180,E1 -12223.719,E2 -12223.719} C_VEL
LIN {X 0,Y 376.104,Z 163.132,A -85,B 0,C 180,E1 -12227.043,E2 -12227.043} C_VEL
LIN {X 0,Y 376.113,Z 163.134,A -85,B 0,C 180,E1 -12230.319,E2 -12230.319} C_VEL
LIN {X 0,Y 376.198,Z 163.123,A -85,B 0,C 180,E1 -12233.565,E2 -12233.565} C_VEL
LIN {X 0,Y 376.338,Z 163.109,A -85,B 0,C 180,E1 -12237.86,E2 -12237.86} C_VEL
LIN {X 0,Y 376.342,Z 163.105,A -85,B 0,C 180,E1 -12242.141,E2 -12242.141} C_VEL
LIN {X 0,Y 376.191,Z 163.122,A -85,B 0,C 180,E1 -12246.436,E2 -12246.436} C_VEL
LIN {X 0,Y 376.111,Z 163.137,A -85,B 0,C 180,E1 -12249.682,E2 -12249.682} C_VEL
LIN {X 0,Y 376.092,Z 163.138,A -85,B 0,C 180,E1 -12253.658,E2 -12253.658} C_VEL
LIN {X 0,Y 376.035,Z 163.148,A -85,B 0,C 180,E1 -12257.4,E2 -12257.4} C_VEL
LIN {X 0,Y 375.982,Z 163.149,A -85,B 0,C 180,E1 -12260.832,E2 -12260.832} C_VEL
LIN {X 0,Y 375.937,Z 163.153,A -85,B 0,C 180,E1 -12264.286,E2 -12264.286} C_VEL
LIN {X 0,Y 375.911,Z 163.158,A -85,B 0,C 180,E1 -12266.661,E2 -12266.661} C_VEL
LIN {X 0,Y 375.914,Z 163.162,A -85,B 0,C 180,E1 -12269.084,E2 -12269.084} C_VEL
LIN {X 0,Y 375.937,Z 163.155,A -85,B 0,C 180,E1 -12271.564,E2 -12271.564} C_VEL
LIN {X 0,Y 375.977,Z 163.151,A -85,B 0,C 180,E1 -12274.666,E2 -12274.666} C_VEL
LIN {X 0,Y 375.935,Z 163.154,A -85,B 0,C 180,E1 -12278.262,E2 -12278.262} C_VEL
LIN {X 0,Y 375.916,Z 163.156,A -85,B 0,C 180,E1 -12281.597,E2 -12281.597} C_VEL
LIN {X 0,Y 375.924,Z 163.16,A -85,B 0,C 180,E1 -12284.73,E2 -12284.73} C_VEL
LIN {X 0,Y 375.91,Z 163.156,A -85,B 0,C 180,E1 -12287.696,E2 -12287.696} C_VEL
LIN {X 0,Y 375.934,Z 163.158,A -85,B 0,C 180,E1 -12290.533,E2 -12290.533} C_VEL
LIN {X 0,Y 375.955,Z 163.151,A -85,B 0,C 180,E1 -12293.498,E2 -12293.498} C_VEL
LIN {X 0,Y 375.942,Z 163.153,A -85,B 0,C 180,E1 -12295.886,E2 -12295.886} C_VEL
LIN {X 0,Y 375.962,Z 163.155,A -85,B 0,C 180,E1 -12299.686,E2 -12299.686} C_VEL
LIN {X 0,Y 375.968,Z 163.297,A -85,B 0,C 180,E1 -12301.924,E2 -12301.924} C_VEL
LIN {X 0,Y 378.134,Z 173.925,A -85,B 0,C 180,E1 -12304.692,E2 -12304.692} C_VEL
LIN {X 0,Y 379.164,Z 180.077,A -85,B 0,C 180,E1 -12306.224,E2 -12306.224} C_VEL
LIN {X 0,Y 378.286,Z 191.048,A -85,B 0,C 180,E1 -12308.759,E2 -12308.759} C_VEL
LIN {X 0,Y 378.223,Z 192.717,A -85,B 0,C 180,E1 -12309.085,E2 -12309.085} C_VEL
LIN {X 0,Y 382.929,Z 222.055,A -85,B 0,C 180,E1 -12309.954,E2 -12309.954} C_VEL
LIN {X 0,Y 381.547,Z 301.429,A -85,B 0,C 180,E1 -12311.542,E2 -12311.542} C_VEL
LIN {X 0,Y 380.944,Z 314.945,A -85,B 0,C 180,E1 -12312.034,E2 -12312.034} C_VEL
LIN {X 0,Y 380.134,Z 327.725,A -85,B 0,C 180,E1 -12312.724,E2 -12312.724} C_VEL
LIN {X 0,Y 379.317,Z 339.467,A -85,B 0,C 180,E1 -12313.587,E2 -12313.587} C_VEL
LIN {X 0,Y 378.419,Z 350.816,A -85,B 0,C 180,E1 -12314.653,E2 -12314.653} C_VEL
LIN {X 0,Y 377.627,Z 360.797,A -85,B 0,C 180,E1 -12315.827,E2 -12315.827} C_VEL
LIN {X 0,Y 376.683,Z 371.063,A -85,B 0,C 180,E1 -12317.335,E2 -12317.335} C_VEL
LIN {X 0,Y 375.825,Z 379.875,A -85,B 0,C 180,E1 -12318.948,E2 -12318.948} C_VEL
LIN {X 0,Y 375.25,Z 386.893,A -85,B 0,C 180,E1 -12320.567,E2 -12320.567} C_VEL
LIN {X 0,Y 374.81,Z 393.322,A -85,B 0,C 180,E1 -12322.457,E2 -12322.457} C_VEL
LIN {X 0,Y 374.589,Z 397.182,A -85,B 0,C 180,E1 -12323.926,E2 -12323.926} C_VEL
LIN {X 0,Y 374.526,Z 400.661,A -85,B 0,C 180,E1 -12325.694,E2 -12325.694} C_VEL
LIN {X 0,Y 374.434,Z 402.214,A -85,B 0,C 180,E1 -12326.771,E2 -12326.771} C_VEL
LIN {X 0,Y 374.416,Z 403.312,A -85,B 0,C 180,E1 -12327.847,E2 -12327.847} C_VEL
LIN {X 0,Y 374.454,Z 403.999,A -85,B 0,C 180,E1 -12328.923,E2 -12328.923} C_VEL
LIN {X 0,Y 374.489,Z 404.295,A -85,B 0,C 180,E1 -12329.999,E2 -12329.999} C_VEL
LIN {X 0,Y 374.453,Z 404.197,A -85,B 0,C 180,E1 -12331.074,E2 -12331.074} C_VEL
LIN {X 0,Y 374.414,Z 403.663,A -85,B 0,C 180,E1 -12332.15,E2 -12332.15} C_VEL
LIN {X 0,Y 374.558,Z 401.39,A -85,B 0,C 180,E1 -12334.303,E2 -12334.303} C_VEL
LIN {X 0,Y 374.642,Z 398.109,A -85,B 0,C 180,E1 -12336.149,E2 -12336.149} C_VEL
LIN {X 0,Y 375.002,Z 393.188,A -85,B 0,C 180,E1 -12338.079,E2 -12338.079} C_VEL
LIN {X 0,Y 375.547,Z 386.774,A -85,B 0,C 180,E1 -12339.967,E2 -12339.967} C_VEL
LIN {X 0,Y 376.179,Z 379.794,A -85,B 0,C 180,E1 -12341.585,E2 -12341.585} C_VEL
LIN {X 0,Y 377.234,Z 371.052,A -85,B 0,C 180,E1 -12343.191,E2 -12343.191} C_VEL
LIN {X 0,Y 378.174,Z 361.638,A -85,B 0,C 180,E1 -12344.595,E2 -12344.595} C_VEL
LIN {X 0,Y 379.117,Z 351.346,A -85,B 0,C 180,E1 -12345.84,E2 -12345.84} C_VEL
LIN {X 0,Y 380.184,Z 339.958,A -85,B 0,C 180,E1 -12346.925,E2 -12346.925} C_VEL
LIN {X 0,Y 381.328,Z 327.505,A -85,B 0,C 180,E1 -12347.841,E2 -12347.841} C_VEL
LIN {X 0,Y 382.183,Z 314.879,A -85,B 0,C 180,E1 -12348.528,E2 -12348.528} C_VEL
LIN {X 0,Y 382.832,Z 301.636,A -85,B 0,C 180,E1 -12349.016,E2 -12349.016} C_VEL
LIN {X 0,Y 383.341,Z 279.124,A -85,B 0,C 180,E1 -12349.498,E2 -12349.498} C_VEL
LIN {X 0,Y 384.242,Z 221.559,A -85,B 0,C 180,E1 -12350.658,E2 -12350.658} C_VEL
LIN {X 0,Y 380.793,Z 201.54,A -85,B 0,C 180,E1 -12351.309,E2 -12351.309} C_VEL
LIN {X 0,Y 378.858,Z 192.003,A -85,B 0,C 180,E1 -12351.691,E2 -12351.691} C_VEL
LIN {X 0,Y 379.654,Z 181.648,A -85,B 0,C 180,E1 -12354.031,E2 -12354.031} C_VEL
LIN {X 0,Y 378.188,Z 173.161,A -85,B 0,C 180,E1 -12356.189,E2 -12356.189} C_VEL
LIN {X 0,Y 375.945,Z 163.235,A -85,B 0,C 180,E1 -12358.914,E2 -12358.914} C_VEL
LIN {X 0,Y 375.932,Z 163.156,A -85,B 0,C 180,E1 -12361.562,E2 -12361.562} C_VEL
LIN {X 0,Y 375.97,Z 163.154,A -85,B 0,C 180,E1 -12364.664,E2 -12364.664} C_VEL
LIN {X 0,Y 375.928,Z 163.156,A -85,B 0,C 180,E1 -12368.261,E2 -12368.261} C_VEL
LIN {X 0,Y 375.907,Z 163.16,A -85,B 0,C 180,E1 -12371.595,E2 -12371.595} C_VEL
LIN {X 0,Y 375.912,Z 163.158,A -85,B 0,C 180,E1 -12374.728,E2 -12374.728} C_VEL
LIN {X 0,Y 375.899,Z 163.163,A -85,B 0,C 180,E1 -12377.695,E2 -12377.695} C_VEL
LIN {X 0,Y 375.926,Z 163.156,A -85,B 0,C 180,E1 -12380.532,E2 -12380.532} C_VEL
LIN {X 0,Y 375.949,Z 163.157,A -85,B 0,C 180,E1 -12383.496,E2 -12383.496} C_VEL
LIN {X 0,Y 375.948,Z 163.151,A -85,B 0,C 180,E1 -12385.887,E2 -12385.887} C_VEL
LIN {X 0,Y 375.95,Z 163.153,A -85,B 0,C 180,E1 -12389.686,E2 -12389.686} C_VEL
LIN {X 0,Y 375.907,Z 163.156,A -85,B 0,C 180,E1 -12392.134,E2 -12392.134} C_VEL
LIN {X 0,Y 375.956,Z 163.15,A -85,B 0,C 180,E1 -12395.715,E2 -12395.715} C_VEL
LIN {X 0,Y 375.969,Z 163.151,A -85,B 0,C 180,E1 -12399.196,E2 -12399.196} C_VEL
LIN {X 0,Y 376.021,Z 163.145,A -85,B 0,C 180,E1 -12402.599,E2 -12402.599} C_VEL
LIN {X 0,Y 376.078,Z 163.137,A -85,B 0,C 180,E1 -12406.342,E2 -12406.342} C_VEL
LIN {X 0,Y 376.1,Z 163.134,A -85,B 0,C 180,E1 -12410.318,E2 -12410.318} C_VEL
LIN {X 0,Y 376.206,Z 163.119,A -85,B 0,C 180,E1 -12413.564,E2 -12413.564} C_VEL
LIN {X 0,Y 376.328,Z 163.105,A -85,B 0,C 180,E1 -12417.859,E2 -12417.859} C_VEL
LIN {X 0,Y 376.325,Z 163.109,A -85,B 0,C 180,E1 -12422.14,E2 -12422.14} C_VEL
LIN {X 0,Y 376.185,Z 163.122,A -85,B 0,C 180,E1 -12426.663,E2 -12426.663} C_VEL
LIN {X 0,Y 376.095,Z 163.134,A -85,B 0,C 180,E1 -12429.682,E2 -12429.682} C_VEL
LIN {X 0,Y 376.076,Z 163.139,A -85,B 0,C 180,E1 -12433.657,E2 -12433.657} C_VEL
LIN {X 0,Y 376.019,Z 163.146,A -85,B 0,C 180,E1 -12437.4,E2 -12437.4} C_VEL
LIN {X 0,Y 375.966,Z 163.153,A -85,B 0,C 180,E1 -12440.832,E2 -12440.832} C_VEL
LIN {X 0,Y 375.945,Z 163.157,A -85,B 0,C 180,E1 -12444.284,E2 -12444.284} C_VEL
LIN {X 0,Y 375.954,Z 163.36,A -85,B 0,C 180,E1 -12447.559,E2 -12447.559} C_VEL
LIN {X 0,Y 378.292,Z 173.752,A -85,B 0,C 180,E1 -12450.414,E2 -12450.414} C_VEL
LIN {X 0,Y 379.225,Z 179.414,A -85,B 0,C 180,E1 -12451.881,E2 -12451.881} C_VEL
LIN {X 0,Y 379.2,Z 181.813,A -85,B 0,C 180,E1 -12452.393,E2 -12452.393} C_VEL
LIN {X 0,Y 382.934,Z 199.004,A -85,B 0,C 180,E1 -12453.048,E2 -12453.048} C_VEL
LIN {X 0,Y 384.606,Z 208.578,A -85,B 0,C 180,E1 -12453.36,E2 -12453.36} C_VEL
LIN {X 0,Y 382.91,Z 290.227,A -85,B 0,C 180,E1 -12455.016,E2 -12455.016} C_VEL
LIN {X 0,Y 382.374,Z 303.329,A -85,B 0,C 180,E1 -12455.498,E2 -12455.498} C_VEL
LIN {X 0,Y 381.69,Z 314.687,A -85,B 0,C 180,E1 -12456.1,E2 -12456.1} C_VEL
LIN {X 0,Y 380.82,Z 326.357,A -85,B 0,C 180,E1 -12456.923,E2 -12456.923} C_VEL
LIN {X 0,Y 379.774,Z 337.983,A -85,B 0,C 180,E1 -12457.988,E2 -12457.988} C_VEL
LIN {X 0,Y 378.754,Z 347.845,A -85,B 0,C 180,E1 -12459.115,E2 -12459.115} C_VEL
LIN {X 0,Y 377.735,Z 357.785,A -85,B 0,C 180,E1 -12460.523,E2 -12460.523} C_VEL
LIN {X 0,Y 376.809,Z 366.285,A -85,B 0,C 180,E1 -12462.025,E2 -12462.025} C_VEL
LIN {X 0,Y 375.912,Z 374.211,A -85,B 0,C 180,E1 -12463.768,E2 -12463.768} C_VEL
LIN {X 0,Y 375.399,Z 379.9,A -85,B 0,C 180,E1 -12465.349,E2 -12465.349} C_VEL
LIN {X 0,Y 374.97,Z 384.501,A -85,B 0,C 180,E1 -12466.967,E2 -12466.967} C_VEL
LIN {X 0,Y 374.644,Z 388.65,A -85,B 0,C 180,E1 -12468.963,E2 -12468.963} C_VEL
LIN {X 0,Y 374.425,Z 390.674,A -85,B 0,C 180,E1 -12470.346,E2 -12470.346} C_VEL
LIN {X 0,Y 374.259,Z 392.204,A -85,B 0,C 180,E1 -12472.063,E2 -12472.063} C_VEL
LIN {X 0,Y 374.196,Z 392.701,A -85,B 0,C 180,E1 -12473.862,E2 -12473.862} C_VEL
LIN {X 0,Y 374.261,Z 392.03,A -85,B 0,C 180,E1 -12475.714,E2 -12475.714} C_VEL
LIN {X 0,Y 374.377,Z 390.052,A -85,B 0,C 180,E1 -12477.645,E2 -12477.645} C_VEL
LIN {X 0,Y 374.668,Z 386.602,A -85,B 0,C 180,E1 -12479.639,E2 -12479.639} C_VEL
LIN {X 0,Y 374.953,Z 382.439,A -85,B 0,C 180,E1 -12481.325,E2 -12481.325} C_VEL
LIN {X 0,Y 375.374,Z 377.032,A -85,B 0,C 180,E1 -12483,E2 -12483} C_VEL
LIN {X 0,Y 376.036,Z 369.401,A -85,B 0,C 180,E1 -12484.839,E2 -12484.839} C_VEL
LIN {X 0,Y 376.762,Z 361.091,A -85,B 0,C 180,E1 -12486.431,E2 -12486.431} C_VEL
LIN {X 0,Y 377.62,Z 351.752,A -85,B 0,C 180,E1 -12487.861,E2 -12487.861} C_VEL
LIN {X 0,Y 378.582,Z 340.823,A -85,B 0,C 180,E1 -12489.208,E2 -12489.208} C_VEL
LIN {X 0,Y 379.452,Z 330.259,A -85,B 0,C 180,E1 -12490.245,E2 -12490.245} C_VEL
LIN {X 0,Y 380.316,Z 317.712,A -85,B 0,C 180,E1 -12491.203,E2 -12491.203} C_VEL
LIN {X 0,Y 380.946,Z 305.002,A -85,B 0,C 180,E1 -12491.932,E2 -12491.932} C_VEL
LIN {X 0,Y 381.545,Z 291.579,A -85,B 0,C 180,E1 -12492.446,E2 -12492.446} C_VEL
LIN {X 0,Y 381.977,Z 270.883,A -85,B 0,C 180,E1 -12492.899,E2 -12492.899} C_VEL
LIN {X 0,Y 382.952,Z 206.714,A -85,B 0,C 180,E1 -12494.159,E2 -12494.159} C_VEL
LIN {X 0,Y 378.408,Z 181.989,A -85,B 0,C 180,E1 -12494.93,E2 -12494.93} C_VEL
LIN {X 0,Y 378.414,Z 180.574,A -85,B 0,C 180,E1 -12495.16,E2 -12495.16} C_VEL
LIN {X 0,Y 378.46,Z 176.008,A -85,B 0,C 180,E1 -12496.306,E2 -12496.306} C_VEL
LIN {X 0,Y 376.283,Z 164.103,A -85,B 0,C 180,E1 -12499.509,E2 -12499.509} C_VEL
LIN {X 0,Y 376.114,Z 163.146,A -85,B 0,C 180,E1 -12499.912,E2 -12499.912} C_VEL
LIN {X 0,Y 376.208,Z 163.12,A -85,B 0,C 180,E1 -12502.487,E2 -12502.487} C_VEL
LIN {X 0,Y 376.167,Z 163.125,A -85,B 0,C 180,E1 -12504.641,E2 -12504.641} C_VEL
LIN {X 0,Y 376.348,Z 163.108,A -85,B 0,C 180,E1 -12507.861,E2 -12507.861} C_VEL
LIN {X 0,Y 376.291,Z 163.109,A -85,B 0,C 180,E1 -12509.005,E2 -12509.005} C_VEL
LIN {X 0,Y 375.709,Z 163.186,A -85,B 0,C 180,E1 -12509.899,E2 -12509.899} C_VEL
LIN {X 0,Y 372.841,Z 163.541,A -85,B 0,C 180,E1 -12511.352,E2 -12511.352} C_VEL
LIN {X 0,Y 370.315,Z 163.856,A -85,B 0,C 180,E1 -12512.526,E2 -12512.526} C_VEL
LIN {X 0,Y 369.17,Z 164,A -85,B 0,C 180,E1 -12513.436,E2 -12513.436} C_VEL
LIN {X 0,Y 369.049,Z 164.011,A -85,B 0,C 180,E1 -12513.745,E2 -12513.745} C_VEL
LIN {X 0,Y 369.185,Z 163.994,A -85,B 0,C 180,E1 -12516.56,E2 -12516.56} C_VEL
LIN {X 0,Y 369.062,Z 164.012,A -85,B 0,C 180,E1 -12519.869,E2 -12519.869} C_VEL
LIN {X 0,Y 369.036,Z 164.016,A -85,B 0,C 180,E1 -12523.773,E2 -12523.773} C_VEL
LIN {X 0,Y 369,Z 164.019,A -85,B 0,C 180,E1 -12527.769,E2 -12527.769} C_VEL
LIN {X 0,Y 368.928,Z 164.032,A -85,B 0,C 180,E1 -12531.221,E2 -12531.221} C_VEL
LIN {X 0,Y 368.957,Z 164.025,A -85,B 0,C 180,E1 -12534.776,E2 -12534.776} C_VEL
LIN {X 0,Y 368.962,Z 164.028,A -85,B 0,C 180,E1 -12537.204,E2 -12537.204} C_VEL
LIN {X 0,Y 368.929,Z 164.031,A -85,B 0,C 180,E1 -12540.954,E2 -12540.954} C_VEL
LIN {X 0,Y 368.928,Z 164.033,A -85,B 0,C 180,E1 -12545.002,E2 -12545.002} C_VEL
LIN {X 0,Y 368.907,Z 164.032,A -85,B 0,C 180,E1 -12548.641,E2 -12548.641} C_VEL
LIN {X 0,Y 368.88,Z 164.032,A -85,B 0,C 180,E1 -12552.01,E2 -12552.01} C_VEL
LIN {X 0,Y 368.883,Z 164.034,A -85,B 0,C 180,E1 -12555.177,E2 -12555.177} C_VEL
LIN {X 0,Y 368.873,Z 164.034,A -85,B 0,C 180,E1 -12558.177,E2 -12558.177} C_VEL
LIN {X 0,Y 368.879,Z 164.033,A -85,B 0,C 180,E1 -12561.366,E2 -12561.366} C_VEL
LIN {X 0,Y 368.936,Z 164.026,A -85,B 0,C 180,E1 -12565.147,E2 -12565.147} C_VEL
LIN {X 0,Y 368.913,Z 164.029,A -85,B 0,C 180,E1 -12569.046,E2 -12569.046} C_VEL
LIN {X 0,Y 368.916,Z 164.028,A -85,B 0,C 180,E1 -12571.559,E2 -12571.559} C_VEL
LIN {X 0,Y 368.934,Z 164.025,A -85,B 0,C 180,E1 -12575.224,E2 -12575.224} C_VEL
LIN {X 0,Y 368.921,Z 164.028,A -85,B 0,C 180,E1 -12578.981,E2 -12578.981} C_VEL
LIN {X 0,Y 368.992,Z 164.024,A -85,B 0,C 180,E1 -12582.258,E2 -12582.258} C_VEL
LIN {X 0,Y 369.038,Z 164.017,A -85,B 0,C 180,E1 -12586.228,E2 -12586.228} C_VEL
LIN {X 0,Y 369.063,Z 164.014,A -85,B 0,C 180,E1 -12590.132,E2 -12590.132} C_VEL
LIN {X 0,Y 369.159,Z 163.999,A -85,B 0,C 180,E1 -12593.441,E2 -12593.441} C_VEL
LIN {X 0,Y 369.302,Z 163.986,A -85,B 0,C 180,E1 -12597.819,E2 -12597.819} C_VEL
LIN {X 0,Y 369.306,Z 163.981,A -85,B 0,C 180,E1 -12602.182,E2 -12602.182} C_VEL
LIN {X 0,Y 369.153,Z 163.998,A -85,B 0,C 180,E1 -12606.56,E2 -12606.56} C_VEL
LIN {X 0,Y 369.062,Z 164.013,A -85,B 0,C 180,E1 -12609.869,E2 -12609.869} C_VEL
LIN {X 0,Y 369.04,Z 164.016,A -85,B 0,C 180,E1 -12613.772,E2 -12613.772} C_VEL
LIN {X 0,Y 368.994,Z 164.021,A -85,B 0,C 180,E1 -12617.743,E2 -12617.743} C_VEL
LIN {X 0,Y 368.912,Z 164.034,A -85,B 0,C 180,E1 -12621.221,E2 -12621.221} C_VEL
LIN {X 0,Y 368.91,Z 164.029,A -85,B 0,C 180,E1 -12623.874,E2 -12623.874} C_VEL
LIN {X 0,Y 368.858,Z 164.041,A -85,B 0,C 180,E1 -12627.212,E2 -12627.212} C_VEL
LIN {X 0,Y 368.894,Z 164.032,A -85,B 0,C 180,E1 -12629.693,E2 -12629.693} C_VEL
LIN {X 0,Y 368.897,Z 164.032,A -85,B 0,C 180,E1 -12633.539,E2 -12633.539} C_VEL
LIN {X 0,Y 368.898,Z 164.035,A -85,B 0,C 180,E1 -12636.854,E2 -12636.854} C_VEL
LIN {X 0,Y 368.886,Z 164.033,A -85,B 0,C 180,E1 -12640.374,E2 -12640.374} C_VEL
LIN {X 0,Y 368.881,Z 164.032,A -85,B 0,C 180,E1 -12643.615,E2 -12643.615} C_VEL
LIN {X 0,Y 368.887,Z 164.037,A -85,B 0,C 180,E1 -12646.695,E2 -12646.695} C_VEL
LIN {X 0,Y 368.887,Z 164.031,A -85,B 0,C 180,E1 -12649.648,E2 -12649.648} C_VEL
LIN {X 0,Y 368.894,Z 164.032,A -85,B 0,C 180,E1 -12653.147,E2 -12653.147} C_VEL
LIN {X 0,Y 368.887,Z 164.037,A -85,B 0,C 180,E1 -12656.46,E2 -12656.46} C_VEL
LIN {X 0,Y 368.895,Z 164.036,A -85,B 0,C 180,E1 -12660.307,E2 -12660.307} C_VEL
LIN {X 0,Y 368.913,Z 164.164,A -85,B 0,C 180,E1 -12661.635,E2 -12661.635} C_VEL
LIN {X 0,Y 371.092,Z 174.797,A -85,B 0,C 180,E1 -12664.462,E2 -12664.462} C_VEL
LIN {X 0,Y 372.182,Z 181.024,A -85,B 0,C 180,E1 -12666.046,E2 -12666.046} C_VEL
LIN {X 0,Y 371.753,Z 187.117,A -85,B 0,C 180,E1 -12667.49,E2 -12667.49} C_VEL
LIN {X 0,Y 371.317,Z 192.639,A -85,B 0,C 180,E1 -12668.719,E2 -12668.719} C_VEL
LIN {X 0,Y 376.184,Z 223.274,A -85,B 0,C 180,E1 -12669.649,E2 -12669.649} C_VEL
LIN {X 0,Y 374.759,Z 301.023,A -85,B 0,C 180,E1 -12671.231,E2 -12671.231} C_VEL
LIN {X 0,Y 374.136,Z 314.628,A -85,B 0,C 180,E1 -12671.731,E2 -12671.731} C_VEL
LIN {X 0,Y 373.371,Z 326.974,A -85,B 0,C 180,E1 -12672.401,E2 -12672.401} C_VEL
LIN {X 0,Y 372.482,Z 338.849,A -85,B 0,C 180,E1 -12673.277,E2 -12673.277} C_VEL
LIN {X 0,Y 371.523,Z 350.289,A -85,B 0,C 180,E1 -12674.361,E2 -12674.361} C_VEL
LIN {X 0,Y 370.766,Z 359.925,A -85,B 0,C 180,E1 -12675.502,E2 -12675.502} C_VEL
LIN {X 0,Y 369.902,Z 369.051,A -85,B 0,C 180,E1 -12676.82,E2 -12676.82} C_VEL
LIN {X 0,Y 368.961,Z 378.194,A -85,B 0,C 180,E1 -12678.462,E2 -12678.462} C_VEL
LIN {X 0,Y 368.317,Z 385.558,A -85,B 0,C 180,E1 -12680.11,E2 -12680.11} C_VEL
LIN {X 0,Y 367.876,Z 391.449,A -85,B 0,C 180,E1 -12681.761,E2 -12681.761} C_VEL
LIN {X 0,Y 367.566,Z 396.07,A -85,B 0,C 180,E1 -12683.411,E2 -12683.411} C_VEL
LIN {X 0,Y 367.475,Z 398.502,A -85,B 0,C 180,E1 -12684.512,E2 -12684.512} C_VEL
LIN {X 0,Y 367.435,Z 400.489,A -85,B 0,C 180,E1 -12685.611,E2 -12685.611} C_VEL
LIN {X 0,Y 367.354,Z 402.055,A -85,B 0,C 180,E1 -12686.709,E2 -12686.709} C_VEL
LIN {X 0,Y 367.319,Z 403.174,A -85,B 0,C 180,E1 -12687.806,E2 -12687.806} C_VEL
LIN {X 0,Y 367.353,Z 403.872,A -85,B 0,C 180,E1 -12688.903,E2 -12688.903} C_VEL
LIN {X 0,Y 367.39,Z 404.178,A -85,B 0,C 180,E1 -12689.999,E2 -12689.999} C_VEL
LIN {X 0,Y 367.352,Z 404.093,A -85,B 0,C 180,E1 -12691.095,E2 -12691.095} C_VEL
LIN {X 0,Y 367.318,Z 403.579,A -85,B 0,C 180,E1 -12692.192,E2 -12692.192} C_VEL
LIN {X 0,Y 367.467,Z 401.326,A -85,B 0,C 180,E1 -12694.386,E2 -12694.386} C_VEL
LIN {X 0,Y 367.54,Z 398.396,A -85,B 0,C 180,E1 -12696.1,E2 -12696.1} C_VEL
LIN {X 0,Y 367.824,Z 394.692,A -85,B 0,C 180,E1 -12697.685,E2 -12697.685} C_VEL
LIN {X 0,Y 368.245,Z 389.732,A -85,B 0,C 180,E1 -12699.335,E2 -12699.335} C_VEL
LIN {X 0,Y 368.877,Z 383.496,A -85,B 0,C 180,E1 -12700.982,E2 -12700.982} C_VEL
LIN {X 0,Y 369.738,Z 375.731,A -85,B 0,C 180,E1 -12702.625,E2 -12702.625} C_VEL
LIN {X 0,Y 370.915,Z 366.001,A -85,B 0,C 180,E1 -12704.258,E2 -12704.258} C_VEL
LIN {X 0,Y 371.864,Z 355.981,A -85,B 0,C 180,E1 -12705.622,E2 -12705.622} C_VEL
LIN {X 0,Y 372.888,Z 346.095,A -85,B 0,C 180,E1 -12706.702,E2 -12706.702} C_VEL
LIN {X 0,Y 373.926,Z 335.383,A -85,B 0,C 180,E1 -12707.641,E2 -12707.641} C_VEL
LIN {X 0,Y 375.018,Z 322.537,A -85,B 0,C 180,E1 -12708.505,E2 -12708.505} C_VEL
LIN {X 0,Y 375.821,Z 309.502,A -85,B 0,C 180,E1 -12709.136,E2 -12709.136} C_VEL
LIN {X 0,Y 376.33,Z 296.744,A -85,B 0,C 180,E1 -12709.535,E2 -12709.535} C_VEL
LIN {X 0,Y 377.719,Z 222.498,A -85,B 0,C 180,E1 -12711.056,E2 -12711.056} C_VEL
LIN {X 0,Y 374.029,Z 201.096,A -85,B 0,C 180,E1 -12711.777,E2 -12711.777} C_VEL
LIN {X 0,Y 372.136,Z 192.258,A -85,B 0,C 180,E1 -12712.131,E2 -12712.131} C_VEL
LIN {X 0,Y 372.173,Z 190.414,A -85,B 0,C 180,E1 -12712.451,E2 -12712.451} C_VEL
LIN {X 0,Y 372.752,Z 182.981,A -85,B 0,C 180,E1 -12714.208,E2 -12714.208} C_VEL
LIN {X 0,Y 371.271,Z 174.517,A -85,B 0,C 180,E1 -12716.412,E2 -12716.412} C_VEL
LIN {X 0,Y 368.902,Z 164.14,A -85,B 0,C 180,E1 -12719.32,E2 -12719.32} C_VEL
LIN {X 0,Y 368.892,Z 164.031,A -85,B 0,C 180,E1 -12723.041,E2 -12723.041} C_VEL
LIN {X 0,Y 368.905,Z 164.033,A -85,B 0,C 180,E1 -12726.196,E2 -12726.196} C_VEL
LIN {X 0,Y 368.867,Z 164.037,A -85,B 0,C 180,E1 -12728.955,E2 -12728.955} C_VEL
LIN {X 0,Y 368.852,Z 164.038,A -85,B 0,C 180,E1 -12732.004,E2 -12732.004} C_VEL
LIN {X 0,Y 368.865,Z 164.039,A -85,B 0,C 180,E1 -12735.173,E2 -12735.173} C_VEL
LIN {X 0,Y 368.852,Z 164.039,A -85,B 0,C 180,E1 -12738.173,E2 -12738.173} C_VEL
LIN {X 0,Y 368.868,Z 164.036,A -85,B 0,C 180,E1 -12741.365,E2 -12741.365} C_VEL
LIN {X 0,Y 368.922,Z 164.027,A -85,B 0,C 180,E1 -12745.144,E2 -12745.144} C_VEL
LIN {X 0,Y 368.886,Z 164.03,A -85,B 0,C 180,E1 -12749.042,E2 -12749.042} C_VEL
LIN {X 0,Y 368.896,Z 164.031,A -85,B 0,C 180,E1 -12751.556,E2 -12751.556} C_VEL
LIN {X 0,Y 368.911,Z 164.031,A -85,B 0,C 180,E1 -12755.221,E2 -12755.221} C_VEL
LIN {X 0,Y 368.909,Z 164.033,A -85,B 0,C 180,E1 -12758.98,E2 -12758.98} C_VEL
LIN {X 0,Y 368.98,Z 164.02,A -85,B 0,C 180,E1 -12762.256,E2 -12762.256} C_VEL
LIN {X 0,Y 369.026,Z 164.014,A -85,B 0,C 180,E1 -12766.227,E2 -12766.227} C_VEL
LIN {X 0,Y 369.05,Z 164.011,A -85,B 0,C 180,E1 -12770.131,E2 -12770.131} C_VEL
LIN {X 0,Y 369.166,Z 163.996,A -85,B 0,C 180,E1 -12773.441,E2 -12773.441} C_VEL
LIN {X 0,Y 369.292,Z 163.981,A -85,B 0,C 180,E1 -12777.818,E2 -12777.818} C_VEL
LIN {X 0,Y 369.289,Z 163.986,A -85,B 0,C 180,E1 -12782.181,E2 -12782.181} C_VEL
LIN {X 0,Y 369.156,Z 163.999,A -85,B 0,C 180,E1 -12786.648,E2 -12786.648} C_VEL
LIN {X 0,Y 369.045,Z 164.013,A -85,B 0,C 180,E1 -12789.868,E2 -12789.868} C_VEL
LIN {X 0,Y 369.024,Z 164.017,A -85,B 0,C 180,E1 -12793.772,E2 -12793.772} C_VEL
LIN {X 0,Y 368.978,Z 164.024,A -85,B 0,C 180,E1 -12797.743,E2 -12797.743} C_VEL
LIN {X 0,Y 368.896,Z 164.034,A -85,B 0,C 180,E1 -12801.221,E2 -12801.221} C_VEL
LIN {X 0,Y 368.905,Z 164.035,A -85,B 0,C 180,E1 -12803.878,E2 -12803.878} C_VEL
LIN {X 0,Y 368.908,Z 164.253,A -85,B 0,C 180,E1 -12807.146,E2 -12807.146} C_VEL
LIN {X 0,Y 371.309,Z 174.756,A -85,B 0,C 180,E1 -12810.104,E2 -12810.104} C_VEL
LIN {X 0,Y 372.358,Z 181.513,A -85,B 0,C 180,E1 -12811.863,E2 -12811.863} C_VEL
LIN {X 0,Y 372.681,Z 183.283,A -85,B 0,C 180,E1 -12812,E2 -12812} C_VEL
LIN {X 0,Y 376.614,Z 201.067,A -85,B 0,C 180,E1 -12812.675,E2 -12812.675} C_VEL
LIN {X 0,Y 378.069,Z 209.862,A -85,B 0,C 180,E1 -12812.964,E2 -12812.964} C_VEL
LIN {X 0,Y 376.324,Z 289.707,A -85,B 0,C 180,E1 -12814.606,E2 -12814.606} C_VEL
LIN {X 0,Y 375.751,Z 303.006,A -85,B 0,C 180,E1 -12815.096,E2 -12815.096} C_VEL
LIN {X 0,Y 375.012,Z 315.2,A -85,B 0,C 180,E1 -12815.754,E2 -12815.754} C_VEL
LIN {X 0,Y 374.048,Z 327.478,A -85,B 0,C 180,E1 -12816.654,E2 -12816.654} C_VEL
LIN {X 0,Y 372.993,Z 338.445,A -85,B 0,C 180,E1 -12817.689,E2 -12817.689} C_VEL
LIN {X 0,Y 371.885,Z 348.403,A -85,B 0,C 180,E1 -12818.856,E2 -12818.856} C_VEL
LIN {X 0,Y 370.949,Z 357.067,A -85,B 0,C 180,E1 -12820.102,E2 -12820.102} C_VEL
LIN {X 0,Y 369.929,Z 365.975,A -85,B 0,C 180,E1 -12821.677,E2 -12821.677} C_VEL
LIN {X 0,Y 369.06,Z 373.268,A -85,B 0,C 180,E1 -12823.278,E2 -12823.278} C_VEL
LIN {X 0,Y 368.406,Z 379.873,A -85,B 0,C 180,E1 -12825.105,E2 -12825.105} C_VEL
LIN {X 0,Y 367.999,Z 384.024,A -85,B 0,C 180,E1 -12826.568,E2 -12826.568} C_VEL
LIN {X 0,Y 367.689,Z 387.63,A -85,B 0,C 180,E1 -12828.197,E2 -12828.197} C_VEL
LIN {X 0,Y 367.382,Z 390.377,A -85,B 0,C 180,E1 -12829.924,E2 -12829.924} C_VEL
LIN {X 0,Y 367.188,Z 392.111,A -85,B 0,C 180,E1 -12831.696,E2 -12831.696} C_VEL
